LIN {X 0,Y 234.885,Z 274.225,A -85,B 0,C 180,E1 -19755.899,E2 -19755.899} C_VEL
LIN {X 0,Y 234.884,Z 274.226,A -85,B 0,C 180,E1 -19758.832,E2 -19758.832} C_VEL
LIN {X 0,Y 234.922,Z 274.22,A -85,B 0,C 180,E1 -19761.079,E2 -19761.079} C_VEL
LIN {X 0,Y 234.962,Z 274.217,A -85,B 0,C 180,E1 -19765.367,E2 -19765.367} C_VEL
LIN {X 0,Y 234.972,Z 274.217,A -85,B 0,C 180,E1 -19770.157,E2 -19770.157} C_VEL
LIN {X 0,Y 234.997,Z 274.213,A -85,B 0,C 180,E1 -19773.794,E2 -19773.794} C_VEL
LIN {X 0,Y 234.993,Z 274.213,A -85,B 0,C 180,E1 -19778.968,E2 -19778.968} C_VEL
LIN {X 0,Y 235.066,Z 274.203,A -85,B 0,C 180,E1 -19783.086,E2 -19783.086} C_VEL
LIN {X 0,Y 235.112,Z 274.196,A -85,B 0,C 180,E1 -19787.922,E2 -19787.922} C_VEL
LIN {X 0,Y 235.325,Z 274.173,A -85,B 0,C 180,E1 -19791.412,E2 -19791.412} C_VEL
LIN {X 0,Y 235.361,Z 274.167,A -85,B 0,C 180,E1 -19793.14,E2 -19793.14} C_VEL
LIN {X 0,Y 235.581,Z 274.14,A -85,B 0,C 180,E1 -19798.29,E2 -19798.29} C_VEL
LIN {X 0,Y 235.598,Z 274.136,A -85,B 0,C 180,E1 -19801.709,E2 -19801.709} C_VEL
LIN {X 0,Y 235.37,Z 274.166,A -85,B 0,C 180,E1 -19806.86,E2 -19806.86} C_VEL
LIN {X 0,Y 235.217,Z 274.185,A -85,B 0,C 180,E1 -19810.327,E2 -19810.327} C_VEL
LIN {X 0,Y 235.116,Z 274.196,A -85,B 0,C 180,E1 -19815.606,E2 -19815.606} C_VEL
LIN {X 0,Y 235.01,Z 274.209,A -85,B 0,C 180,E1 -19819.205,E2 -19819.205} C_VEL
LIN {X 0,Y 234.942,Z 274.219,A -85,B 0,C 180,E1 -19822.885,E2 -19822.885} C_VEL
LIN {X 0,Y 234.931,Z 274.22,A -85,B 0,C 180,E1 -19826.662,E2 -19826.662} C_VEL
LIN {X 0,Y 234.9,Z 274.225,A -85,B 0,C 180,E1 -19830.572,E2 -19830.572} C_VEL
LIN {X 0,Y 234.927,Z 274.224,A -85,B 0,C 180,E1 -19834.639,E2 -19834.639} C_VEL
LIN {X 0,Y 234.963,Z 274.311,A -85,B 0,C 180,E1 -19838.638,E2 -19838.638} C_VEL
LIN {X 0,Y 235.52,Z 277.972,A -85,B 0,C 180,E1 -19843.34,E2 -19843.34} C_VEL
LIN {X 0,Y 236.021,Z 280.862,A -85,B 0,C 180,E1 -19846.774,E2 -19846.774} C_VEL
LIN {X 0,Y 236.594,Z 284.553,A -85,B 0,C 180,E1 -19850.896,E2 -19850.896} C_VEL
LIN {X 0,Y 235.974,Z 285.513,A -85,B 0,C 180,E1 -19851.81,E2 -19851.81} C_VEL
LIN {X 0,Y 233.129,Z 287.277,A -85,B 0,C 180,E1 -19853.227,E2 -19853.227} C_VEL
LIN {X 0,Y 230.118,Z 289.077,A -85,B 0,C 180,E1 -19854.673,E2 -19854.673} C_VEL
LIN {X 0,Y 229.294,Z 290.098,A -85,B 0,C 180,E1 -19855.624,E2 -19855.624} C_VEL
LIN {X 0,Y 228.939,Z 291.784,A -85,B 0,C 180,E1 -19857.204,E2 -19857.204} C_VEL
LIN {X 0,Y 229.832,Z 294.982,A -85,B 0,C 180,E1 -19857.512,E2 -19857.512} C_VEL
LIN {X 0,Y 233.461,Z 307.701,A -85,B 0,C 180,E1 -19858.946,E2 -19858.946} C_VEL
LIN {X 0,Y 235.843,Z 319.474,A -85,B 0,C 180,E1 -19860.432,E2 -19860.432} C_VEL
LIN {X 0,Y 237.308,Z 330.805,A -85,B 0,C 180,E1 -19862.06,E2 -19862.06} C_VEL
LIN {X 0,Y 237.836,Z 342.077,A -85,B 0,C 180,E1 -19863.924,E2 -19863.924} C_VEL
LIN {X 0,Y 237.611,Z 348.307,A -85,B 0,C 180,E1 -19865.071,E2 -19865.071} C_VEL
LIN {X 0,Y 234.977,Z 358.761,A -85,B 0,C 180,E1 -19867.119,E2 -19867.119} C_VEL
LIN {X 0,Y 232.724,Z 367.292,A -85,B 0,C 180,E1 -19869.237,E2 -19869.237} C_VEL
LIN {X 0,Y 230.624,Z 375.499,A -85,B 0,C 180,E1 -19871.798,E2 -19871.798} C_VEL
LIN {X 0,Y 228.803,Z 382.165,A -85,B 0,C 180,E1 -19874.409,E2 -19874.409} C_VEL
LIN {X 0,Y 227.207,Z 388.266,A -85,B 0,C 180,E1 -19877.495,E2 -19877.495} C_VEL
LIN {X 0,Y 226.332,Z 392.236,A -85,B 0,C 180,E1 -19880.166,E2 -19880.166} C_VEL
LIN {X 0,Y 225.809,Z 395.171,A -85,B 0,C 180,E1 -19882.848,E2 -19882.848} C_VEL
LIN {X 0,Y 225.59,Z 397.12,A -85,B 0,C 180,E1 -19885.505,E2 -19885.505} C_VEL
LIN {X 0,Y 225.644,Z 398.178,A -85,B 0,C 180,E1 -19888.215,E2 -19888.215} C_VEL
LIN {X 0,Y 225.716,Z 398.393,A -85,B 0,C 180,E1 -19890,E2 -19890} C_VEL
LIN {X 0,Y 225.642,Z 398.168,A -85,B 0,C 180,E1 -19891.785,E2 -19891.785} C_VEL
LIN {X 0,Y 225.643,Z 396.545,A -85,B 0,C 180,E1 -19895.361,E2 -19895.361} C_VEL
LIN {X 0,Y 225.779,Z 395.136,A -85,B 0,C 180,E1 -19897.152,E2 -19897.152} C_VEL
LIN {X 0,Y 226.332,Z 392.186,A -85,B 0,C 180,E1 -19899.833,E2 -19899.833} C_VEL
LIN {X 0,Y 227.206,Z 388.196,A -85,B 0,C 180,E1 -19902.505,E2 -19902.505} C_VEL
LIN {X 0,Y 228.797,Z 382.068,A -85,B 0,C 180,E1 -19905.591,E2 -19905.591} C_VEL
LIN {X 0,Y 230.624,Z 375.38,A -85,B 0,C 180,E1 -19908.201,E2 -19908.201} C_VEL
LIN {X 0,Y 232.613,Z 368.002,A -85,B 0,C 180,E1 -19910.509,E2 -19910.509} C_VEL
LIN {X 0,Y 235.015,Z 358.578,A -85,B 0,C 180,E1 -19912.877,E2 -19912.877} C_VEL
LIN {X 0,Y 237.592,Z 348.074,A -85,B 0,C 180,E1 -19914.93,E2 -19914.93} C_VEL
LIN {X 0,Y 237.692,Z 338.928,A -85,B 0,C 180,E1 -19916.585,E2 -19916.585} C_VEL
LIN {X 0,Y 237.116,Z 329.199,A -85,B 0,C 180,E1 -19918.134,E2 -19918.134} C_VEL
LIN {X 0,Y 235.415,Z 317.231,A -85,B 0,C 180,E1 -19919.816,E2 -19919.816} C_VEL
LIN {X 0,Y 232.586,Z 304.36,A -85,B 0,C 180,E1 -19921.403,E2 -19921.403} C_VEL
LIN {X 0,Y 229.458,Z 294.179,A -85,B 0,C 180,E1 -19922.535,E2 -19922.535} C_VEL
LIN {X 0,Y 228.907,Z 291.66,A -85,B 0,C 180,E1 -19922.767,E2 -19922.767} C_VEL
LIN {X 0,Y 229.544,Z 288.869,A -85,B 0,C 180,E1 -19925.572,E2 -19925.572} C_VEL
LIN {X 0,Y 229.598,Z 285.783,A -85,B 0,C 180,E1 -19928.866,E2 -19928.866} C_VEL
LIN {X 0,Y 229.109,Z 282.514,A -85,B 0,C 180,E1 -19932.591,E2 -19932.591} C_VEL
LIN {X 0,Y 228.398,Z 278.449,A -85,B 0,C 180,E1 -19937.604,E2 -19937.604} C_VEL
LIN {X 0,Y 227.922,Z 275.092,A -85,B 0,C 180,E1 -19942.314,E2 -19942.314} C_VEL
LIN {X 0,Y 227.879,Z 275.104,A -85,B 0,C 180,E1 -19946.378,E2 -19946.378} C_VEL
LIN {X 0,Y 227.876,Z 275.105,A -85,B 0,C 180,E1 -19950.432,E2 -19950.432} C_VEL
LIN {X 0,Y 227.881,Z 275.103,A -85,B 0,C 180,E1 -19954.42,E2 -19954.42} C_VEL
LIN {X 0,Y 227.952,Z 275.092,A -85,B 0,C 180,E1 -19958.286,E2 -19958.286} C_VEL
LIN {X 0,Y 228.035,Z 275.079,A -85,B 0,C 180,E1 -19962.826,E2 -19962.826} C_VEL
LIN {X 0,Y 228.073,Z 275.075,A -85,B 0,C 180,E1 -19967.543,E2 -19967.543} C_VEL
LIN {X 0,Y 228.265,Z 275.052,A -85,B 0,C 180,E1 -19971.144,E2 -19971.144} C_VEL
LIN {X 0,Y 228.32,Z 275.043,A -85,B 0,C 180,E1 -19972.928,E2 -19972.928} C_VEL
LIN {X 0,Y 228.555,Z 275.011,A -85,B 0,C 180,E1 -19978.238,E2 -19978.238} C_VEL
LIN {X 0,Y 228.54,Z 275.015,A -85,B 0,C 180,E1 -19981.762,E2 -19981.762} C_VEL
LIN {X 0,Y 228.315,Z 275.046,A -85,B 0,C 180,E1 -19987.073,E2 -19987.073} C_VEL
LIN {X 0,Y 228.143,Z 275.068,A -85,B 0,C 180,E1 -19990.651,E2 -19990.651} C_VEL
LIN {X 0,Y 228.042,Z 275.079,A -85,B 0,C 180,E1 -19994.274,E2 -19994.274} C_VEL
LIN {X 0,Y 227.97,Z 275.087,A -85,B 0,C 180,E1 -19997.956,E2 -19997.956} C_VEL
LIN {X 0,Y 227.917,Z 275.095,A -85,B 0,C 180,E1 -20002.32,E2 -20002.32} C_VEL
LIN {X 0,Y 227.945,Z 275.091,A -85,B 0,C 180,E1 -20006.603,E2 -20006.603} C_VEL
LIN {X 0,Y 227.911,Z 275.097,A -85,B 0,C 180,E1 -20010.297,E2 -20010.297} C_VEL
LIN {X 0,Y 227.89,Z 275.098,A -85,B 0,C 180,E1 -20013.719,E2 -20013.719} C_VEL
LIN {X 0,Y 227.849,Z 275.105,A -85,B 0,C 180,E1 -20018.09,E2 -20018.09} C_VEL
LIN {X 0,Y 227.806,Z 275.106,A -85,B 0,C 180,E1 -20022.744,E2 -20022.744} C_VEL
LIN {X 0,Y 227.793,Z 275.112,A -85,B 0,C 180,E1 -20027.253,E2 -20027.253} C_VEL
LIN {X 0,Y 227.794,Z 275.111,A -85,B 0,C 180,E1 -20027.771,E2 -20027.771} C_VEL
LIN {X 0,Y 228.121,Z 277.722,A -85,B 0,C 180,E1 -20031.963,E2 -20031.963} C_VEL
LIN {X 0,Y 228.132,Z 279.267,A -85,B 0,C 180,E1 -20034.174,E2 -20034.174} C_VEL
LIN {X 0,Y 227.974,Z 281.488,A -85,B 0,C 180,E1 -20037.173,E2 -20037.173} C_VEL
LIN {X 0,Y 229.009,Z 284.65,A -85,B 0,C 180,E1 -20037.516,E2 -20037.516} C_VEL
LIN {X 0,Y 233.392,Z 296.608,A -85,B 0,C 180,E1 -20039.049,E2 -20039.049} C_VEL
LIN {X 0,Y 236.369,Z 307.22,A -85,B 0,C 180,E1 -20040.527,E2 -20040.527} C_VEL
LIN {X 0,Y 238.446,Z 317.934,A -85,B 0,C 180,E1 -20042.157,E2 -20042.157} C_VEL
LIN {X 0,Y 239.698,Z 328.159,A -85,B 0,C 180,E1 -20043.909,E2 -20043.909} C_VEL
LIN {X 0,Y 239.776,Z 330.767,A -85,B 0,C 180,E1 -20044.384,E2 -20044.384} C_VEL
LIN {X 0,Y 237.493,Z 341.214,A -85,B 0,C 180,E1 -20046.223,E2 -20046.223} C_VEL
LIN {X 0,Y 235.276,Z 350.46,A -85,B 0,C 180,E1 -20048.263,E2 -20048.263} C_VEL
LIN {X 0,Y 232.951,Z 358.989,A -85,B 0,C 180,E1 -20050.618,E2 -20050.618} C_VEL
LIN {X 0,Y 230.753,Z 366.396,A -85,B 0,C 180,E1 -20053.182,E2 -20053.182} C_VEL
LIN {X 0,Y 229.031,Z 372.336,A -85,B 0,C 180,E1 -20055.79,E2 -20055.79} C_VEL
LIN {X 0,Y 227.7,Z 377.028,A -85,B 0,C 180,E1 -20058.427,E2 -20058.427} C_VEL
LIN {X 0,Y 226.773,Z 380.616,A -85,B 0,C 180,E1 -20061.086,E2 -20061.086} C_VEL
LIN {X 0,Y 226.101,Z 383.466,A -85,B 0,C 180,E1 -20064.086,E2 -20064.086} C_VEL
LIN {X 0,Y 225.853,Z 384.85,A -85,B 0,C 180,E1 -20066.432,E2 -20066.432} C_VEL
LIN {X 0,Y 225.747,Z 385.686,A -85,B 0,C 180,E1 -20070,E2 -20070} C_VEL
LIN {X 0,Y 225.75,Z 385.493,A -85,B 0,C 180,E1 -20071.784,E2 -20071.784} C_VEL
LIN {X 0,Y 225.853,Z 384.907,A -85,B 0,C 180,E1 -20073.568,E2 -20073.568} C_VEL
LIN {X 0,Y 226.335,Z 382.583,A -85,B 0,C 180,E1 -20077.135,E2 -20077.135} C_VEL
LIN {X 0,Y 227.072,Z 379.715,A -85,B 0,C 180,E1 -20079.801,E2 -20079.801} C_VEL
LIN {X 0,Y 228.089,Z 375.825,A -85,B 0,C 180,E1 -20082.456,E2 -20082.456} C_VEL
LIN {X 0,Y 229.547,Z 370.804,A -85,B 0,C 180,E1 -20085.085,E2 -20085.085} C_VEL
LIN {X 0,Y 231.365,Z 364.48,A -85,B 0,C 180,E1 -20087.684,E2 -20087.684} C_VEL
LIN {X 0,Y 233.685,Z 356.561,A -85,B 0,C 180,E1 -20090.234,E2 -20090.234} C_VEL
LIN {X 0,Y 235.646,Z 349.088,A -85,B 0,C 180,E1 -20092.195,E2 -20092.195} C_VEL
LIN {X 0,Y 237.852,Z 339.709,A -85,B 0,C 180,E1 -20094.204,E2 -20094.204} C_VEL
LIN {X 0,Y 239.901,Z 330.235,A -85,B 0,C 180,E1 -20095.835,E2 -20095.835} C_VEL
LIN {X 0,Y 238.792,Z 319.781,A -85,B 0,C 180,E1 -20097.674,E2 -20097.674} C_VEL
LIN {X 0,Y 236.677,Z 308.483,A -85,B 0,C 180,E1 -20099.435,E2 -20099.435} C_VEL
LIN {X 0,Y 234.207,Z 299.118,A -85,B 0,C 180,E1 -20100.756,E2 -20100.756} C_VEL
LIN {X 0,Y 230.069,Z 287.427,A -85,B 0,C 180,E1 -20102.302,E2 -20102.302} C_VEL
LIN {X 0,Y 227.94,Z 281.449,A -85,B 0,C 180,E1 -20103.022,E2 -20103.022} C_VEL
LIN {X 0,Y 228.147,Z 278.702,A -85,B 0,C 180,E1 -20106.781,E2 -20106.781} C_VEL
LIN {X 0,Y 227.963,Z 276.309,A -85,B 0,C 180,E1 -20110.348,E2 -20110.348} C_VEL
LIN {X 0,Y 227.796,Z 275.113,A -85,B 0,C 180,E1 -20112.23,E2 -20112.23} C_VEL
LIN {X 0,Y 227.824,Z 275.102,A -85,B 0,C 180,E1 -20115.196,E2 -20115.196} C_VEL
LIN {X 0,Y 227.827,Z 275.105,A -85,B 0,C 180,E1 -20119.623,E2 -20119.623} C_VEL
LIN {X 0,Y 227.901,Z 275.098,A -85,B 0,C 180,E1 -20124.132,E2 -20124.132} C_VEL
LIN {X 0,Y 227.874,Z 275.097,A -85,B 0,C 180,E1 -20128.378,E2 -20128.378} C_VEL
LIN {X 0,Y 227.888,Z 275.094,A -85,B 0,C 180,E1 -20132.445,E2 -20132.445} C_VEL
LIN {X 0,Y 227.909,Z 275.09,A -85,B 0,C 180,E1 -20136.367,E2 -20136.367} C_VEL
LIN {X 0,Y 227.927,Z 275.092,A -85,B 0,C 180,E1 -20140.173,E2 -20140.173} C_VEL
LIN {X 0,Y 228.032,Z 275.08,A -85,B 0,C 180,E1 -20143.896,E2 -20143.896} C_VEL
LIN {X 0,Y 228.069,Z 275.075,A -85,B 0,C 180,E1 -20147.543,E2 -20147.543} C_VEL
LIN {X 0,Y 228.263,Z 275.052,A -85,B 0,C 180,E1 -20151.144,E2 -20151.144} C_VEL
LIN {X 0,Y 228.313,Z 275.046,A -85,B 0,C 180,E1 -20152.927,E2 -20152.927} C_VEL
LIN {X 0,Y 228.54,Z 275.017,A -85,B 0,C 180,E1 -20158.238,E2 -20158.238} C_VEL
LIN {X 0,Y 228.556,Z 275.013,A -85,B 0,C 180,E1 -20161.762,E2 -20161.762} C_VEL
LIN {X 0,Y 228.321,Z 275.043,A -85,B 0,C 180,E1 -20167.072,E2 -20167.072} C_VEL
LIN {X 0,Y 228.148,Z 275.067,A -85,B 0,C 180,E1 -20170.651,E2 -20170.651} C_VEL
LIN {X 0,Y 228.067,Z 275.077,A -85,B 0,C 180,E1 -20174.272,E2 -20174.272} C_VEL
LIN {X 0,Y 228.005,Z 275.083,A -85,B 0,C 180,E1 -20177.953,E2 -20177.953} C_VEL
LIN {X 0,Y 227.92,Z 275.095,A -85,B 0,C 180,E1 -20182.321,E2 -20182.321} C_VEL
LIN {X 0,Y 227.908,Z 275.094,A -85,B 0,C 180,E1 -20186.584,E2 -20186.584} C_VEL
LIN {X 0,Y 227.875,Z 275.101,A -85,B 0,C 180,E1 -20190.28,E2 -20190.28} C_VEL
LIN {X 0,Y 227.878,Z 275.102,A -85,B 0,C 180,E1 -20193.72,E2 -20193.72} C_VEL
LIN {X 0,Y 227.952,Z 275.294,A -85,B 0,C 180,E1 -20198.07,E2 -20198.07} C_VEL
LIN {X 0,Y 228.451,Z 278.676,A -85,B 0,C 180,E1 -20202.594,E2 -20202.594} C_VEL
LIN {X 0,Y 228.782,Z 280.62,A -85,B 0,C 180,E1 -20205.045,E2 -20205.045} C_VEL
LIN {X 0,Y 229.307,Z 283.762,A -85,B 0,C 180,E1 -20208.78,E2 -20208.78} C_VEL
LIN {X 0,Y 229.621,Z 286.876,A -85,B 0,C 180,E1 -20212.255,E2 -20212.255} C_VEL
LIN {X 0,Y 229.555,Z 288.921,A -85,B 0,C 180,E1 -20214.43,E2 -20214.43} C_VEL
LIN {X 0,Y 229.294,Z 290.098,A -85,B 0,C 180,E1 -20215.624,E2 -20215.624} C_VEL
LIN {X 0,Y 229.334,Z 291.506,A -85,B 0,C 180,E1 -20216.361,E2 -20216.361} C_VEL
LIN {X 0,Y 229.683,Z 294.528,A -85,B 0,C 180,E1 -20217.107,E2 -20217.107} C_VEL
LIN {X 0,Y 230.101,Z 299.741,A -85,B 0,C 180,E1 -20217.804,E2 -20217.804} C_VEL
LIN {X 0,Y 229.759,Z 306.045,A -85,B 0,C 180,E1 -20218.259,E2 -20218.259} C_VEL
LIN {X 0,Y 228.821,Z 314.395,A -85,B 0,C 180,E1 -20218.89,E2 -20218.89} C_VEL
LIN {X 0,Y 228.994,Z 318.121,A -85,B 0,C 180,E1 -20219.328,E2 -20219.328} C_VEL
LIN {X 0,Y 230.539,Z 329.644,A -85,B 0,C 180,E1 -20221.03,E2 -20221.03} C_VEL
LIN {X 0,Y 231.175,Z 340.556,A -85,B 0,C 180,E1 -20222.869,E2 -20222.869} C_VEL
LIN {X 0,Y 231.134,Z 348.109,A -85,B 0,C 180,E1 -20224.323,E2 -20224.323} C_VEL
LIN {X 0,Y 228.449,Z 358.564,A -85,B 0,C 180,E1 -20226.426,E2 -20226.426} C_VEL
LIN {X 0,Y 225.753,Z 368.275,A -85,B 0,C 180,E1 -20228.943,E2 -20228.943} C_VEL
LIN {X 0,Y 223.867,Z 375.3,A -85,B 0,C 180,E1 -20231.229,E2 -20231.229} C_VEL
LIN {X 0,Y 221.929,Z 381.966,A -85,B 0,C 180,E1 -20233.913,E2 -20233.913} C_VEL
LIN {X 0,Y 220.226,Z 388.066,A -85,B 0,C 180,E1 -20237.092,E2 -20237.092} C_VEL
LIN {X 0,Y 219.318,Z 392.036,A -85,B 0,C 180,E1 -20239.849,E2 -20239.849} C_VEL
LIN {X 0,Y 218.736,Z 394.971,A -85,B 0,C 180,E1 -20242.616,E2 -20242.616} C_VEL
LIN {X 0,Y 218.488,Z 397.091,A -85,B 0,C 180,E1 -20245.685,E2 -20245.685} C_VEL
LIN {X 0,Y 218.541,Z 397.979,A -85,B 0,C 180,E1 -20248.157,E2 -20248.157} C_VEL
LIN {X 0,Y 218.631,Z 398.194,A -85,B 0,C 180,E1 -20250,E2 -20250} C_VEL
LIN {X 0,Y 218.539,Z 397.968,A -85,B 0,C 180,E1 -20251.843,E2 -20251.843} C_VEL
LIN {X 0,Y 218.484,Z 397.08,A -85,B 0,C 180,E1 -20254.302,E2 -20254.302} C_VEL
LIN {X 0,Y 218.709,Z 394.935,A -85,B 0,C 180,E1 -20257.385,E2 -20257.385} C_VEL
LIN {X 0,Y 219.317,Z 391.984,A -85,B 0,C 180,E1 -20260.151,E2 -20260.151} C_VEL
LIN {X 0,Y 220.226,Z 387.994,A -85,B 0,C 180,E1 -20262.908,E2 -20262.908} C_VEL
LIN {X 0,Y 221.922,Z 381.865,A -85,B 0,C 180,E1 -20266.087,E2 -20266.087} C_VEL
LIN {X 0,Y 223.873,Z 375.177,A -85,B 0,C 180,E1 -20268.77,E2 -20268.77} C_VEL
LIN {X 0,Y 226.172,Z 366.906,A -85,B 0,C 180,E1 -20271.407,E2 -20271.407} C_VEL
LIN {X 0,Y 228.459,Z 358.375,A -85,B 0,C 180,E1 -20273.573,E2 -20273.573} C_VEL
LIN {X 0,Y 231.076,Z 347.868,A -85,B 0,C 180,E1 -20275.684,E2 -20275.684} C_VEL
LIN {X 0,Y 231.009,Z 337.161,A -85,B 0,C 180,E1 -20277.682,E2 -20277.682} C_VEL
LIN {X 0,Y 230.172,Z 326.464,A -85,B 0,C 180,E1 -20279.414,E2 -20279.414} C_VEL
LIN {X 0,Y 228.497,Z 315.557,A -85,B 0,C 180,E1 -20280.978,E2 -20280.978} C_VEL
LIN {X 0,Y 225.642,Z 303.453,A -85,B 0,C 180,E1 -20282.537,E2 -20282.537} C_VEL
LIN {X 0,Y 222.241,Z 292.284,A -85,B 0,C 180,E1 -20283.822,E2 -20283.822} C_VEL
LIN {X 0,Y 222.151,Z 291.412,A -85,B 0,C 180,E1 -20283.927,E2 -20283.927} C_VEL
LIN {X 0,Y 222.571,Z 288.652,A -85,B 0,C 180,E1 -20286.866,E2 -20286.866} C_VEL
LIN {X 0,Y 222.562,Z 286.597,A -85,B 0,C 180,E1 -20289.165,E2 -20289.165} C_VEL
LIN {X 0,Y 221.977,Z 283.153,A -85,B 0,C 180,E1 -20293.264,E2 -20293.264} C_VEL
LIN {X 0,Y 221.325,Z 279.326,A -85,B 0,C 180,E1 -20298.176,E2 -20298.176} C_VEL
LIN {X 0,Y 220.864,Z 275.998,A -85,B 0,C 180,E1 -20302.866,E2 -20302.866} C_VEL
LIN {X 0,Y 220.812,Z 275.984,A -85,B 0,C 180,E1 -20307.243,E2 -20307.243} C_VEL
LIN {X 0,Y 220.801,Z 275.985,A -85,B 0,C 180,E1 -20311.481,E2 -20311.481} C_VEL
LIN {X 0,Y 220.833,Z 275.98,A -85,B 0,C 180,E1 -20315.561,E2 -20315.561} C_VEL
LIN {X 0,Y 220.884,Z 275.972,A -85,B 0,C 180,E1 -20319.513,E2 -20319.513} C_VEL
LIN {X 0,Y 221.017,Z 275.955,A -85,B 0,C 180,E1 -20323.37,E2 -20323.37} C_VEL
LIN {X 0,Y 221.012,Z 275.953,A -85,B 0,C 180,E1 -20327.139,E2 -20327.139} C_VEL
LIN {X 0,Y 221.203,Z 275.93,A -85,B 0,C 180,E1 -20330.859,E2 -20330.859} C_VEL
LIN {X 0,Y 221.138,Z 275.937,A -85,B 0,C 180,E1 -20334.529,E2 -20334.529} C_VEL
LIN {X 0,Y 221.513,Z 275.889,A -85,B 0,C 180,E1 -20338.182,E2 -20338.182} C_VEL
LIN {X 0,Y 221.474,Z 275.895,A -85,B 0,C 180,E1 -20341.819,E2 -20341.819} C_VEL
LIN {X 0,Y 221.252,Z 275.924,A -85,B 0,C 180,E1 -20347.3,E2 -20347.3} C_VEL
LIN {X 0,Y 221.064,Z 275.948,A -85,B 0,C 180,E1 -20350.997,E2 -20350.997} C_VEL
LIN {X 0,Y 220.992,Z 275.958,A -85,B 0,C 180,E1 -20356.632,E2 -20356.632} C_VEL
LIN {X 0,Y 220.877,Z 275.972,A -85,B 0,C 180,E1 -20360.488,E2 -20360.488} C_VEL
LIN {X 0,Y 220.863,Z 275.973,A -85,B 0,C 180,E1 -20364.436,E2 -20364.436} C_VEL
LIN {X 0,Y 220.839,Z 275.976,A -85,B 0,C 180,E1 -20368.513,E2 -20368.513} C_VEL
LIN {X 0,Y 220.825,Z 275.978,A -85,B 0,C 180,E1 -20372.755,E2 -20372.755} C_VEL
LIN {X 0,Y 220.839,Z 275.976,A -85,B 0,C 180,E1 -20377.288,E2 -20377.288} C_VEL
LIN {X 0,Y 220.768,Z 275.984,A -85,B 0,C 180,E1 -20381.953,E2 -20381.953} C_VEL
LIN {X 0,Y 220.763,Z 275.987,A -85,B 0,C 180,E1 -20385.543,E2 -20385.543} C_VEL
LIN {X 0,Y 220.751,Z 275.989,A -85,B 0,C 180,E1 -20387.075,E2 -20387.075} C_VEL
LIN {X 0,Y 221.057,Z 277.949,A -85,B 0,C 180,E1 -20390.517,E2 -20390.517} C_VEL
LIN {X 0,Y 221.13,Z 279.485,A -85,B 0,C 180,E1 -20392.853,E2 -20392.853} C_VEL
LIN {X 0,Y 221.021,Z 281.838,A -85,B 0,C 180,E1 -20396.007,E2 -20396.007} C_VEL
LIN {X 0,Y 222.261,Z 285.131,A -85,B 0,C 180,E1 -20396.415,E2 -20396.415} C_VEL
LIN {X 0,Y 226.389,Z 296.266,A -85,B 0,C 180,E1 -20397.93,E2 -20397.93} C_VEL
LIN {X 0,Y 229.522,Z 306.734,A -85,B 0,C 180,E1 -20399.475,E2 -20399.475} C_VEL
LIN {X 0,Y 231.762,Z 318.117,A -85,B 0,C 180,E1 -20401.276,E2 -20401.276} C_VEL
LIN {X 0,Y 233.027,Z 328.374,A -85,B 0,C 180,E1 -20403.103,E2 -20403.103} C_VEL
LIN {X 0,Y 233.117,Z 332.258,A -85,B 0,C 180,E1 -20403.838,E2 -20403.838} C_VEL
LIN {X 0,Y 230.757,Z 342.47,A -85,B 0,C 180,E1 -20405.722,E2 -20405.722} C_VEL
LIN {X 0,Y 228.615,Z 350.944,A -85,B 0,C 180,E1 -20407.676,E2 -20407.676} C_VEL
LIN {X 0,Y 226.266,Z 359.191,A -85,B 0,C 180,E1 -20410.022,E2 -20410.022} C_VEL
LIN {X 0,Y 223.971,Z 366.597,A -85,B 0,C 180,E1 -20412.657,E2 -20412.657} C_VEL
LIN {X 0,Y 222.157,Z 372.537,A -85,B 0,C 180,E1 -20415.34,E2 -20415.34} C_VEL
LIN {X 0,Y 220.745,Z 377.229,A -85,B 0,C 180,E1 -20418.057,E2 -20418.057} C_VEL
LIN {X 0,Y 219.773,Z 380.817,A -85,B 0,C 180,E1 -20420.8,E2 -20420.8} C_VEL
LIN {X 0,Y 219,Z 383.876,A -85,B 0,C 180,E1 -20424.174,E2 -20424.174} C_VEL
LIN {X 0,Y 218.765,Z 385.05,A -85,B 0,C 180,E1 -20426.316,E2 -20426.316} C_VEL
LIN {X 0,Y 218.67,Z 385.657,A -85,B 0,C 180,E1 -20428.158,E2 -20428.158} C_VEL
LIN {X 0,Y 218.662,Z 385.885,A -85,B 0,C 180,E1 -20430,E2 -20430} C_VEL
LIN {X 0,Y 218.67,Z 385.692,A -85,B 0,C 180,E1 -20431.842,E2 -20431.842} C_VEL
LIN {X 0,Y 218.765,Z 385.106,A -85,B 0,C 180,E1 -20433.684,E2 -20433.684} C_VEL
LIN {X 0,Y 219.045,Z 383.886,A -85,B 0,C 180,E1 -20435.939,E2 -20435.939} C_VEL
LIN {X 0,Y 219.783,Z 380.969,A -85,B 0,C 180,E1 -20439.2,E2 -20439.2} C_VEL
LIN {X 0,Y 220.718,Z 377.438,A -85,B 0,C 180,E1 -20441.945,E2 -20441.945} C_VEL
LIN {X 0,Y 222.13,Z 372.802,A -85,B 0,C 180,E1 -20444.662,E2 -20444.662} C_VEL
LIN {X 0,Y 224.248,Z 365.812,A -85,B 0,C 180,E1 -20447.793,E2 -20447.793} C_VEL
LIN {X 0,Y 226.609,Z 358.229,A -85,B 0,C 180,E1 -20450.421,E2 -20450.421} C_VEL
LIN {X 0,Y 228.953,Z 349.809,A -85,B 0,C 180,E1 -20452.739,E2 -20452.739} C_VEL
LIN {X 0,Y 231.384,Z 339.905,A -85,B 0,C 180,E1 -20454.926,E2 -20454.926} C_VEL
LIN {X 0,Y 233.29,Z 331.717,A -85,B 0,C 180,E1 -20456.382,E2 -20456.382} C_VEL
LIN {X 0,Y 232.431,Z 322.328,A -85,B 0,C 180,E1 -20458.131,E2 -20458.131} C_VEL
LIN {X 0,Y 230.553,Z 311.378,A -85,B 0,C 180,E1 -20459.958,E2 -20459.958} C_VEL
LIN {X 0,Y 228.018,Z 301.264,A -85,B 0,C 180,E1 -20461.49,E2 -20461.49} C_VEL
LIN {X 0,Y 223.748,Z 288.775,A -85,B 0,C 180,E1 -20463.25,E2 -20463.25} C_VEL
LIN {X 0,Y 221.095,Z 282.49,A -85,B 0,C 180,E1 -20464.1,E2 -20464.1} C_VEL
LIN {X 0,Y 220.947,Z 281.662,A -85,B 0,C 180,E1 -20464.206,E2 -20464.206} C_VEL
LIN {X 0,Y 221.134,Z 279.434,A -85,B 0,C 180,E1 -20467.388,E2 -20467.388} C_VEL
LIN {X 0,Y 220.985,Z 277.582,A -85,B 0,C 180,E1 -20470.246,E2 -20470.246} C_VEL
LIN {X 0,Y 220.752,Z 275.981,A -85,B 0,C 180,E1 -20472.925,E2 -20472.925} C_VEL
LIN {X 0,Y 220.763,Z 275.985,A -85,B 0,C 180,E1 -20477.072,E2 -20477.072} C_VEL
LIN {X 0,Y 220.808,Z 275.98,A -85,B 0,C 180,E1 -20480.463,E2 -20480.463} C_VEL
LIN {X 0,Y 220.826,Z 275.976,A -85,B 0,C 180,E1 -20482.793,E2 -20482.793} C_VEL
LIN {X 0,Y 220.826,Z 275.978,A -85,B 0,C 180,E1 -20487.245,E2 -20487.245} C_VEL
LIN {X 0,Y 220.839,Z 275.976,A -85,B 0,C 180,E1 -20491.487,E2 -20491.487} C_VEL
LIN {X 0,Y 220.865,Z 275.971,A -85,B 0,C 180,E1 -20495.565,E2 -20495.565} C_VEL
LIN {X 0,Y 220.879,Z 275.972,A -85,B 0,C 180,E1 -20499.512,E2 -20499.512} C_VEL
LIN {X 0,Y 220.993,Z 275.958,A -85,B 0,C 180,E1 -20503.368,E2 -20503.368} C_VEL
LIN {X 0,Y 221.068,Z 275.948,A -85,B 0,C 180,E1 -20509.004,E2 -20509.004} C_VEL
LIN {X 0,Y 221.25,Z 275.926,A -85,B 0,C 180,E1 -20512.7,E2 -20512.7} C_VEL
LIN {X 0,Y 221.473,Z 275.897,A -85,B 0,C 180,E1 -20518.181,E2 -20518.181} C_VEL
LIN {X 0,Y 221.514,Z 275.89,A -85,B 0,C 180,E1 -20521.818,E2 -20521.818} C_VEL
LIN {X 0,Y 221.257,Z 275.922,A -85,B 0,C 180,E1 -20527.299,E2 -20527.299} C_VEL
LIN {X 0,Y 221.07,Z 275.948,A -85,B 0,C 180,E1 -20530.996,E2 -20530.996} C_VEL
LIN {X 0,Y 220.998,Z 275.955,A -85,B 0,C 180,E1 -20534.739,E2 -20534.739} C_VEL
LIN {X 0,Y 220.923,Z 275.966,A -85,B 0,C 180,E1 -20538.549,E2 -20538.549} C_VEL
LIN {X 0,Y 220.866,Z 275.972,A -85,B 0,C 180,E1 -20542.662,E2 -20542.662} C_VEL
LIN {X 0,Y 220.854,Z 275.973,A -85,B 0,C 180,E1 -20546.999,E2 -20546.999} C_VEL
LIN {X 0,Y 220.82,Z 275.979,A -85,B 0,C 180,E1 -20550.758,E2 -20550.758} C_VEL
LIN {X 0,Y 220.795,Z 275.984,A -85,B 0,C 180,E1 -20554.956,E2 -20554.956} C_VEL
LIN {X 0,Y 220.894,Z 276.177,A -85,B 0,C 180,E1 -20557.306,E2 -20557.306} C_VEL
LIN {X 0,Y 221.348,Z 279.408,A -85,B 0,C 180,E1 -20561.818,E2 -20561.818} C_VEL
LIN {X 0,Y 221.988,Z 283.216,A -85,B 0,C 180,E1 -20566.733,E2 -20566.733} C_VEL
LIN {X 0,Y 222.562,Z 286.651,A -85,B 0,C 180,E1 -20570.835,E2 -20570.835} C_VEL
LIN {X 0,Y 222.54,Z 289.729,A -85,B 0,C 180,E1 -20574.251,E2 -20574.251} C_VEL
LIN {X 0,Y 222.147,Z 291.448,A -85,B 0,C 180,E1 -20576.055,E2 -20576.055} C_VEL
LIN {X 0,Y 223.067,Z 294.804,A -85,B 0,C 180,E1 -20576.401,E2 -20576.401} C_VEL
LIN {X 0,Y 226.676,Z 307.124,A -85,B 0,C 180,E1 -20577.876,E2 -20577.876} C_VEL
LIN {X 0,Y 228.994,Z 318.121,A -85,B 0,C 180,E1 -20579.328,E2 -20579.328} C_VEL
LIN {X 0,Y 229.149,Z 323.436,A -85,B 0,C 180,E1 -20579.988,E2 -20579.988} C_VEL
LIN {X 0,Y 227.421,Z 332.31,A -85,B 0,C 180,E1 -20581.007,E2 -20581.007} C_VEL
LIN {X 0,Y 225.179,Z 340.906,A -85,B 0,C 180,E1 -20582.173,E2 -20582.173} C_VEL
LIN {X 0,Y 224.568,Z 345.73,A -85,B 0,C 180,E1 -20583.054,E2 -20583.054} C_VEL
LIN {X 0,Y 224.196,Z 350.215,A -85,B 0,C 180,E1 -20583.968,E2 -20583.968} C_VEL
LIN {X 0,Y 221.402,Z 360.16,A -85,B 0,C 180,E1 -20586.126,E2 -20586.126} C_VEL
LIN {X 0,Y 218.657,Z 369.706,A -85,B 0,C 180,E1 -20588.766,E2 -20588.766} C_VEL
LIN {X 0,Y 216.748,Z 376.338,A -85,B 0,C 180,E1 -20591.08,E2 -20591.08} C_VEL
LIN {X 0,Y 214.811,Z 382.762,A -85,B 0,C 180,E1 -20593.853,E2 -20593.853} C_VEL
LIN {X 0,Y 213.261,Z 387.866,A -85,B 0,C 180,E1 -20596.662,E2 -20596.662} C_VEL
LIN {X 0,Y 212.304,Z 391.836,A -85,B 0,C 180,E1 -20599.509,E2 -20599.509} C_VEL
LIN {X 0,Y 211.67,Z 394.771,A -85,B 0,C 180,E1 -20602.368,E2 -20602.368} C_VEL
LIN {X 0,Y 211.393,Z 397.026,A -85,B 0,C 180,E1 -20605.855,E2 -20605.855} C_VEL
LIN {X 0,Y 211.442,Z 397.779,A -85,B 0,C 180,E1 -20608.095,E2 -20608.095} C_VEL
LIN {X 0,Y 211.547,Z 397.994,A -85,B 0,C 180,E1 -20610,E2 -20610} C_VEL
LIN {X 0,Y 211.44,Z 397.767,A -85,B 0,C 180,E1 -20611.905,E2 -20611.905} C_VEL
LIN {X 0,Y 211.487,Z 396.144,A -85,B 0,C 180,E1 -20615.721,E2 -20615.721} C_VEL
LIN {X 0,Y 211.65,Z 394.734,A -85,B 0,C 180,E1 -20617.633,E2 -20617.633} C_VEL
LIN {X 0,Y 212.304,Z 391.783,A -85,B 0,C 180,E1 -20620.49,E2 -20620.49} C_VEL
LIN {X 0,Y 213.26,Z 387.791,A -85,B 0,C 180,E1 -20623.337,E2 -20623.337} C_VEL
LIN {X 0,Y 215.085,Z 381.663,A -85,B 0,C 180,E1 -20626.613,E2 -20626.613} C_VEL
LIN {X 0,Y 217.151,Z 374.975,A -85,B 0,C 180,E1 -20629.374,E2 -20629.374} C_VEL
LIN {X 0,Y 219.43,Z 367.056,A -85,B 0,C 180,E1 -20631.981,E2 -20631.981} C_VEL
LIN {X 0,Y 221.962,Z 358.172,A -85,B 0,C 180,E1 -20634.307,E2 -20634.307} C_VEL
LIN {X 0,Y 224.422,Z 348.841,A -85,B 0,C 180,E1 -20636.253,E2 -20636.253} C_VEL
LIN {X 0,Y 224.461,Z 338.049,A -85,B 0,C 180,E1 -20638.367,E2 -20638.367} C_VEL
LIN {X 0,Y 223.681,Z 327.455,A -85,B 0,C 180,E1 -20640.18,E2 -20640.18} C_VEL
LIN {X 0,Y 221.863,Z 315.531,A -85,B 0,C 180,E1 -20641.988,E2 -20641.988} C_VEL
LIN {X 0,Y 218.944,Z 303.041,A -85,B 0,C 180,E1 -20643.676,E2 -20643.676} C_VEL
LIN {X 0,Y 215.359,Z 291.471,A -85,B 0,C 180,E1 -20645.084,E2 -20645.084} C_VEL
LIN {X 0,Y 215.543,Z 289.456,A -85,B 0,C 180,E1 -20647.1,E2 -20647.1} C_VEL
LIN {X 0,Y 215.335,Z 286.357,A -85,B 0,C 180,E1 -20650.749,E2 -20650.749} C_VEL
LIN {X 0,Y 214.875,Z 283.776,A -85,B 0,C 180,E1 -20653.982,E2 -20653.982} C_VEL
LIN {X 0,Y 214.277,Z 280.043,A -85,B 0,C 180,E1 -20659.006,E2 -20659.006} C_VEL
LIN {X 0,Y 213.79,Z 276.856,A -85,B 0,C 180,E1 -20663.83,E2 -20663.83} C_VEL
LIN {X 0,Y 213.768,Z 276.863,A -85,B 0,C 180,E1 -20668.737,E2 -20668.737} C_VEL
LIN {X 0,Y 213.784,Z 276.859,A -85,B 0,C 180,E1 -20672.597,E2 -20672.597} C_VEL
LIN {X 0,Y 213.808,Z 276.854,A -85,B 0,C 180,E1 -20676.981,E2 -20676.981} C_VEL
LIN {X 0,Y 213.944,Z 276.835,A -85,B 0,C 180,E1 -20682.804,E2 -20682.804} C_VEL
LIN {X 0,Y 213.954,Z 276.831,A -85,B 0,C 180,E1 -20686.707,E2 -20686.707} C_VEL
LIN {X 0,Y 214.141,Z 276.81,A -85,B 0,C 180,E1 -20690.555,E2 -20690.555} C_VEL
LIN {X 0,Y 214.099,Z 276.814,A -85,B 0,C 180,E1 -20694.349,E2 -20694.349} C_VEL
LIN {X 0,Y 214.446,Z 276.769,A -85,B 0,C 180,E1 -20698.122,E2 -20698.122} C_VEL
LIN {X 0,Y 214.541,Z 276.76,A -85,B 0,C 180,E1 -20700,E2 -20700} C_VEL
LIN {X 0,Y 214.411,Z 276.775,A -85,B 0,C 180,E1 -20701.878,E2 -20701.878} C_VEL
LIN {X 0,Y 214.192,Z 276.803,A -85,B 0,C 180,E1 -20707.542,E2 -20707.542} C_VEL
LIN {X 0,Y 213.995,Z 276.826,A -85,B 0,C 180,E1 -20711.365,E2 -20711.365} C_VEL
LIN {X 0,Y 213.91,Z 276.837,A -85,B 0,C 180,E1 -20715.239,E2 -20715.239} C_VEL
LIN {X 0,Y 213.82,Z 276.85,A -85,B 0,C 180,E1 -20719.189,E2 -20719.189} C_VEL
LIN {X 0,Y 213.812,Z 276.851,A -85,B 0,C 180,E1 -20723.231,E2 -20723.231} C_VEL
LIN {X 0,Y 213.83,Z 276.848,A -85,B 0,C 180,E1 -20727.45,E2 -20727.45} C_VEL
LIN {X 0,Y 213.78,Z 276.855,A -85,B 0,C 180,E1 -20731.736,E2 -20731.736} C_VEL
LIN {X 0,Y 213.749,Z 276.861,A -85,B 0,C 180,E1 -20736.288,E2 -20736.288} C_VEL
LIN {X 0,Y 213.712,Z 276.865,A -85,B 0,C 180,E1 -20741.126,E2 -20741.126} C_VEL
LIN {X 0,Y 213.704,Z 276.867,A -85,B 0,C 180,E1 -20743.68,E2 -20743.68} C_VEL
LIN {X 0,Y 213.702,Z 276.865,A -85,B 0,C 180,E1 -20746.345,E2 -20746.345} C_VEL
LIN {X 0,Y 213.93,Z 278.279,A -85,B 0,C 180,E1 -20749.077,E2 -20749.077} C_VEL
LIN {X 0,Y 214.106,Z 280.085,A -85,B 0,C 180,E1 -20751.981,E2 -20751.981} C_VEL
LIN {X 0,Y 214.038,Z 281.886,A -85,B 0,C 180,E1 -20754.701,E2 -20754.701} C_VEL
LIN {X 0,Y 215.214,Z 285.229,A -85,B 0,C 180,E1 -20755.15,E2 -20755.15} C_VEL
LIN {X 0,Y 218.702,Z 293.765,A -85,B 0,C 180,E1 -20756.407,E2 -20756.407} C_VEL
LIN {X 0,Y 222.22,Z 304.734,A -85,B 0,C 180,E1 -20758.091,E2 -20758.091} C_VEL
LIN {X 0,Y 224.483,Z 314.476,A -85,B 0,C 180,E1 -20759.68,E2 -20759.68} C_VEL
LIN {X 0,Y 226.04,Z 325.148,A -85,B 0,C 180,E1 -20761.583,E2 -20761.583} C_VEL
LIN {X 0,Y 226.625,Z 332.467,A -85,B 0,C 180,E1 -20763.029,E2 -20763.029} C_VEL
LIN {X 0,Y 224.298,Z 342.674,A -85,B 0,C 180,E1 -20764.976,E2 -20764.976} C_VEL
LIN {X 0,Y 221.912,Z 351.68,A -85,B 0,C 180,E1 -20767.125,E2 -20767.125} C_VEL
LIN {X 0,Y 219.195,Z 360.74,A -85,B 0,C 180,E1 -20769.838,E2 -20769.838} C_VEL
LIN {X 0,Y 216.85,Z 367.909,A -85,B 0,C 180,E1 -20772.555,E2 -20772.555} C_VEL
LIN {X 0,Y 215.302,Z 372.738,A -85,B 0,C 180,E1 -20774.862,E2 -20774.862} C_VEL
LIN {X 0,Y 213.797,Z 377.431,A -85,B 0,C 180,E1 -20777.663,E2 -20777.663} C_VEL
LIN {X 0,Y 212.752,Z 381.018,A -85,B 0,C 180,E1 -20780.493,E2 -20780.493} C_VEL
LIN {X 0,Y 212.244,Z 382.87,A -85,B 0,C 180,E1 -20782.389,E2 -20782.389} C_VEL
LIN {X 0,Y 211.893,Z 384.261,A -85,B 0,C 180,E1 -20784.29,E2 -20784.29} C_VEL
LIN {X 0,Y 211.592,Z 385.857,A -85,B 0,C 180,E1 -20788.097,E2 -20788.097} C_VEL
LIN {X 0,Y 211.579,Z 386.084,A -85,B 0,C 180,E1 -20790,E2 -20790} C_VEL
LIN {X 0,Y 211.592,Z 385.891,A -85,B 0,C 180,E1 -20791.904,E2 -20791.904} C_VEL
LIN {X 0,Y 211.893,Z 384.339,A -85,B 0,C 180,E1 -20795.711,E2 -20795.711} C_VEL
LIN {X 0,Y 212.245,Z 382.982,A -85,B 0,C 180,E1 -20797.611,E2 -20797.611} C_VEL
LIN {X 0,Y 213.058,Z 380.114,A -85,B 0,C 180,E1 -20800.453,E2 -20800.453} C_VEL
LIN {X 0,Y 214.223,Z 376.223,A -85,B 0,C 180,E1 -20803.277,E2 -20803.277} C_VEL
LIN {X 0,Y 215.844,Z 371.202,A -85,B 0,C 180,E1 -20806.067,E2 -20806.067} C_VEL
LIN {X 0,Y 217.894,Z 364.875,A -85,B 0,C 180,E1 -20808.817,E2 -20808.817} C_VEL
LIN {X 0,Y 220.431,Z 356.955,A -85,B 0,C 180,E1 -20811.51,E2 -20811.51} C_VEL
LIN {X 0,Y 222.701,Z 348.739,A -85,B 0,C 180,E1 -20813.768,E2 -20813.768} C_VEL
LIN {X 0,Y 225.227,Z 339.036,A -85,B 0,C 180,E1 -20815.904,E2 -20815.904} C_VEL
LIN {X 0,Y 226.7,Z 333.2,A -85,B 0,C 180,E1 -20816.962,E2 -20816.962} C_VEL
LIN {X 0,Y 225.904,Z 323.555,A -85,B 0,C 180,E1 -20818.853,E2 -20818.853} C_VEL
LIN {X 0,Y 224.108,Z 312.646,A -85,B 0,C 180,E1 -20820.771,E2 -20820.771} C_VEL
LIN {X 0,Y 221.973,Z 303.727,A -85,B 0,C 180,E1 -20822.215,E2 -20822.215} C_VEL
LIN {X 0,Y 217.702,Z 291.17,A -85,B 0,C 180,E1 -20824.13,E2 -20824.13} C_VEL
LIN {X 0,Y 214.939,Z 284.788,A -85,B 0,C 180,E1 -20825.087,E2 -20825.087} C_VEL
LIN {X 0,Y 213.996,Z 281.885,A -85,B 0,C 180,E1 -20825.478,E2 -20825.478} C_VEL
LIN {X 0,Y 214.077,Z 279.834,A -85,B 0,C 180,E1 -20828.591,E2 -20828.591} C_VEL
LIN {X 0,Y 213.917,Z 278.295,A -85,B 0,C 180,E1 -20831.078,E2 -20831.078} C_VEL
LIN {X 0,Y 213.704,Z 276.86,A -85,B 0,C 180,E1 -20833.68,E2 -20833.68} C_VEL
LIN {X 0,Y 213.705,Z 276.864,A -85,B 0,C 180,E1 -20836.345,E2 -20836.345} C_VEL
LIN {X 0,Y 213.736,Z 276.86,A -85,B 0,C 180,E1 -20841.336,E2 -20841.336} C_VEL
LIN {X 0,Y 213.77,Z 276.855,A -85,B 0,C 180,E1 -20846.02,E2 -20846.02} C_VEL
LIN {X 0,Y 213.783,Z 276.855,A -85,B 0,C 180,E1 -20850.454,E2 -20850.454} C_VEL
LIN {X 0,Y 213.801,Z 276.852,A -85,B 0,C 180,E1 -20854.701,E2 -20854.701} C_VEL
LIN {X 0,Y 213.8,Z 276.853,A -85,B 0,C 180,E1 -20858.802,E2 -20858.802} C_VEL
LIN {X 0,Y 213.924,Z 276.836,A -85,B 0,C 180,E1 -20862.802,E2 -20862.802} C_VEL
LIN {X 0,Y 213.946,Z 276.835,A -85,B 0,C 180,E1 -20866.706,E2 -20866.706} C_VEL
LIN {X 0,Y 214.14,Z 276.81,A -85,B 0,C 180,E1 -20870.555,E2 -20870.555} C_VEL
LIN {X 0,Y 214.086,Z 276.816,A -85,B 0,C 180,E1 -20874.348,E2 -20874.348} C_VEL
LIN {X 0,Y 214.41,Z 276.777,A -85,B 0,C 180,E1 -20878.122,E2 -20878.122} C_VEL
LIN {X 0,Y 214.517,Z 276.763,A -85,B 0,C 180,E1 -20880,E2 -20880} C_VEL
LIN {X 0,Y 214.447,Z 276.77,A -85,B 0,C 180,E1 -20881.878,E2 -20881.878} C_VEL
LIN {X 0,Y 214.197,Z 276.801,A -85,B 0,C 180,E1 -20887.541,E2 -20887.541} C_VEL
LIN {X 0,Y 214.001,Z 276.827,A -85,B 0,C 180,E1 -20891.364,E2 -20891.364} C_VEL
LIN {X 0,Y 213.936,Z 276.834,A -85,B 0,C 180,E1 -20895.237,E2 -20895.237} C_VEL
LIN {X 0,Y 213.839,Z 276.847,A -85,B 0,C 180,E1 -20899.187,E2 -20899.187} C_VEL
LIN {X 0,Y 213.801,Z 276.852,A -85,B 0,C 180,E1 -20903.232,E2 -20903.232} C_VEL
LIN {X 0,Y 213.786,Z 276.855,A -85,B 0,C 180,E1 -20907.426,E2 -20907.426} C_VEL
LIN {X 0,Y 213.76,Z 276.861,A -85,B 0,C 180,E1 -20911.739,E2 -20911.739} C_VEL
LIN {X 0,Y 213.795,Z 276.929,A -85,B 0,C 180,E1 -20916.278,E2 -20916.278} C_VEL
LIN {X 0,Y 214.295,Z 280.142,A -85,B 0,C 180,E1 -20921.035,E2 -20921.035} C_VEL
LIN {X 0,Y 214.895,Z 283.85,A -85,B 0,C 180,E1 -20926.013,E2 -20926.013} C_VEL
LIN {X 0,Y 215.343,Z 286.415,A -85,B 0,C 180,E1 -20929.252,E2 -20929.252} C_VEL
LIN {X 0,Y 215.549,Z 289.511,A -85,B 0,C 180,E1 -20932.901,E2 -20932.901} C_VEL
LIN {X 0,Y 215.353,Z 291.268,A -85,B 0,C 180,E1 -20934.838,E2 -20934.838} C_VEL
LIN {X 0,Y 216.336,Z 294.63,A -85,B 0,C 180,E1 -20935.211,E2 -20935.211} C_VEL
LIN {X 0,Y 219.824,Z 306.297,A -85,B 0,C 180,E1 -20936.693,E2 -20936.693} C_VEL
LIN {X 0,Y 222.377,Z 318.047,A -85,B 0,C 180,E1 -20938.327,E2 -20938.327} C_VEL
LIN {X 0,Y 223.936,Z 329.473,A -85,B 0,C 180,E1 -20940.095,E2 -20940.095} C_VEL
LIN {X 0,Y 224.575,Z 340.351,A -85,B 0,C 180,E1 -20942.003,E2 -20942.003} C_VEL
LIN {X 0,Y 224.568,Z 345.73,A -85,B 0,C 180,E1 -20943.054,E2 -20943.054} C_VEL
LIN {X 0,Y 224.06,Z 348.886,A -85,B 0,C 180,E1 -20943.661,E2 -20943.661} C_VEL
LIN {X 0,Y 222.041,Z 353.464,A -85,B 0,C 180,E1 -20944.469,E2 -20944.469} C_VEL
LIN {X 0,Y 215.086,Z 363.326,A -85,B 0,C 180,E1 -20946.356,E2 -20946.356} C_VEL
LIN {X 0,Y 212.764,Z 367.286,A -85,B 0,C 180,E1 -20947.382,E2 -20947.382} C_VEL
LIN {X 0,Y 212.286,Z 368.558,A -85,B 0,C 180,E1 -20947.772,E2 -20947.772} C_VEL
LIN {X 0,Y 210.027,Z 376.139,A -85,B 0,C 180,E1 -20950.45,E2 -20950.45} C_VEL
LIN {X 0,Y 207.953,Z 382.562,A -85,B 0,C 180,E1 -20953.305,E2 -20953.305} C_VEL
LIN {X 0,Y 206.314,Z 387.665,A -85,B 0,C 180,E1 -20956.205,E2 -20956.205} C_VEL
LIN {X 0,Y 205.283,Z 391.636,A -85,B 0,C 180,E1 -20959.146,E2 -20959.146} C_VEL
LIN {X 0,Y 204.626,Z 394.572,A -85,B 0,C 180,E1 -20962.103,E2 -20962.103} C_VEL
LIN {X 0,Y 204.398,Z 395.969,A -85,B 0,C 180,E1 -20964.079,E2 -20964.079} C_VEL
LIN {X 0,Y 204.345,Z 397.579,A -85,B 0,C 180,E1 -20968.029,E2 -20968.029} C_VEL
LIN {X 0,Y 204.465,Z 397.795,A -85,B 0,C 180,E1 -20970,E2 -20970} C_VEL
LIN {X 0,Y 204.343,Z 397.567,A -85,B 0,C 180,E1 -20971.971,E2 -20971.971} C_VEL
LIN {X 0,Y 204.394,Z 395.943,A -85,B 0,C 180,E1 -20975.921,E2 -20975.921} C_VEL
LIN {X 0,Y 204.611,Z 394.533,A -85,B 0,C 180,E1 -20977.897,E2 -20977.897} C_VEL
LIN {X 0,Y 205.282,Z 391.581,A -85,B 0,C 180,E1 -20980.853,E2 -20980.853} C_VEL
LIN {X 0,Y 206.313,Z 387.589,A -85,B 0,C 180,E1 -20983.795,E2 -20983.795} C_VEL
LIN {X 0,Y 208.279,Z 381.462,A -85,B 0,C 180,E1 -20987.173,E2 -20987.173} C_VEL
LIN {X 0,Y 210.46,Z 374.774,A -85,B 0,C 180,E1 -20990.016,E2 -20990.016} C_VEL
LIN {X 0,Y 212.897,Z 366.587,A -85,B 0,C 180,E1 -20992.784,E2 -20992.784} C_VEL
LIN {X 0,Y 215.48,Z 357.968,A -85,B 0,C 180,E1 -20995.087,E2 -20995.087} C_VEL
LIN {X 0,Y 217.776,Z 349.784,A -85,B 0,C 180,E1 -20996.859,E2 -20996.859} C_VEL
LIN {X 0,Y 217.952,Z 339.844,A -85,B 0,C 180,E1 -20998.926,E2 -20998.926} C_VEL
LIN {X 0,Y 217.288,Z 329.024,A -85,B 0,C 180,E1 -21000.894,E2 -21000.894} C_VEL
LIN {X 0,Y 215.86,Z 318.507,A -85,B 0,C 180,E1 -21002.601,E2 -21002.601} C_VEL
LIN {X 0,Y 213.167,Z 305.978,A -85,B 0,C 180,E1 -21004.433,E2 -21004.433} C_VEL
LIN {X 0,Y 209.678,Z 294.671,A -85,B 0,C 180,E1 -21005.976,E2 -21005.976} C_VEL
LIN {X 0,Y 208.547,Z 291.464,A -85,B 0,C 180,E1 -21006.397,E2 -21006.397} C_VEL
LIN {X 0,Y 208.488,Z 290.981,A -85,B 0,C 180,E1 -21006.481,E2 -21006.481} C_VEL
LIN {X 0,Y 208.383,Z 288.17,A -85,B 0,C 180,E1 -21009.852,E2 -21009.852} C_VEL
LIN {X 0,Y 208.054,Z 286.112,A -85,B 0,C 180,E1 -21012.5,E2 -21012.5} C_VEL
LIN {X 0,Y 207.444,Z 282.527,A -85,B 0,C 180,E1 -21017.345,E2 -21017.345} C_VEL
LIN {X 0,Y 206.977,Z 279.176,A -85,B 0,C 180,E1 -21022.324,E2 -21022.324} C_VEL
LIN {X 0,Y 206.729,Z 277.737,A -85,B 0,C 180,E1 -21024.694,E2 -21024.694} C_VEL
LIN {X 0,Y 206.695,Z 277.743,A -85,B 0,C 180,E1 -21029.334,E2 -21029.334} C_VEL
LIN {X 0,Y 206.696,Z 277.744,A -85,B 0,C 180,E1 -21033.767,E2 -21033.767} C_VEL
LIN {X 0,Y 206.734,Z 277.735,A -85,B 0,C 180,E1 -21038.041,E2 -21038.041} C_VEL
LIN {X 0,Y 206.873,Z 277.716,A -85,B 0,C 180,E1 -21042.197,E2 -21042.197} C_VEL
LIN {X 0,Y 206.896,Z 277.711,A -85,B 0,C 180,E1 -21046.244,E2 -21046.244} C_VEL
LIN {X 0,Y 207.1,Z 277.687,A -85,B 0,C 180,E1 -21050.231,E2 -21050.231} C_VEL
LIN {X 0,Y 207.06,Z 277.691,A -85,B 0,C 180,E1 -21054.156,E2 -21054.156} C_VEL
LIN {X 0,Y 207.383,Z 277.649,A -85,B 0,C 180,E1 -21058.058,E2 -21058.058} C_VEL
LIN {X 0,Y 207.506,Z 277.637,A -85,B 0,C 180,E1 -21060,E2 -21060} C_VEL
LIN {X 0,Y 207.054,Z 277.692,A -85,B 0,C 180,E1 -21063.893,E2 -21063.893} C_VEL
LIN {X 0,Y 207.136,Z 277.681,A -85,B 0,C 180,E1 -21067.8,E2 -21067.8} C_VEL
LIN {X 0,Y 206.918,Z 277.707,A -85,B 0,C 180,E1 -21071.759,E2 -21071.759} C_VEL
LIN {X 0,Y 206.844,Z 277.717,A -85,B 0,C 180,E1 -21075.773,E2 -21075.773} C_VEL
LIN {X 0,Y 206.858,Z 277.717,A -85,B 0,C 180,E1 -21077.955,E2 -21077.955} C_VEL
LIN {X 0,Y 206.755,Z 277.73,A -85,B 0,C 180,E1 -21083.396,E2 -21083.396} C_VEL
LIN {X 0,Y 206.746,Z 277.732,A -85,B 0,C 180,E1 -21088.419,E2 -21088.419} C_VEL
LIN {X 0,Y 206.71,Z 277.736,A -85,B 0,C 180,E1 -21092.956,E2 -21092.956} C_VEL
LIN {X 0,Y 206.723,Z 277.735,A -85,B 0,C 180,E1 -21095.32,E2 -21095.32} C_VEL
LIN {X 0,Y 206.664,Z 277.739,A -85,B 0,C 180,E1 -21100.251,E2 -21100.251} C_VEL
LIN {X 0,Y 206.631,Z 277.747,A -85,B 0,C 180,E1 -21105.583,E2 -21105.583} C_VEL
LIN {X 0,Y 206.946,Z 279.968,A -85,B 0,C 180,E1 -21109.816,E2 -21109.816} C_VEL
LIN {X 0,Y 207.045,Z 282.157,A -85,B 0,C 180,E1 -21113.346,E2 -21113.346} C_VEL
LIN {X 0,Y 208.125,Z 285.237,A -85,B 0,C 180,E1 -21113.763,E2 -21113.763} C_VEL
LIN {X 0,Y 210.764,Z 290.973,A -85,B 0,C 180,E1 -21114.708,E2 -21114.708} C_VEL
LIN {X 0,Y 214.269,Z 300.794,A -85,B 0,C 180,E1 -21116.287,E2 -21116.287} C_VEL
LIN {X 0,Y 217.306,Z 311.953,A -85,B 0,C 180,E1 -21118.183,E2 -21118.183} C_VEL
LIN {X 0,Y 219.149,Z 322.908,A -85,B 0,C 180,E1 -21120.173,E2 -21120.173} C_VEL
LIN {X 0,Y 220.033,Z 332.68,A -85,B 0,C 180,E1 -21122.152,E2 -21122.152} C_VEL
LIN {X 0,Y 219.875,Z 335.126,A -85,B 0,C 180,E1 -21122.647,E2 -21122.647} C_VEL
LIN {X 0,Y 217.325,Z 344.832,A -85,B 0,C 180,E1 -21124.629,E2 -21124.629} C_VEL
LIN {X 0,Y 214.835,Z 353.659,A -85,B 0,C 180,E1 -21126.886,E2 -21126.886} C_VEL
LIN {X 0,Y 212.13,Z 362.269,A -85,B 0,C 180,E1 -21129.643,E2 -21129.643} C_VEL
LIN {X 0,Y 209.71,Z 369.137,A -85,B 0,C 180,E1 -21132.445,E2 -21132.445} C_VEL
LIN {X 0,Y 207.883,Z 374.63,A -85,B 0,C 180,E1 -21135.312,E2 -21135.312} C_VEL
LIN {X 0,Y 206.442,Z 378.94,A -85,B 0,C 180,E1 -21138.214,E2 -21138.214} C_VEL
LIN {X 0,Y 205.742,Z 381.219,A -85,B 0,C 180,E1 -21140.166,E2 -21140.166} C_VEL
LIN {X 0,Y 205.202,Z 383.071,A -85,B 0,C 180,E1 -21142.126,E2 -21142.126} C_VEL
LIN {X 0,Y 204.771,Z 384.667,A -85,B 0,C 180,E1 -21144.457,E2 -21144.457} C_VEL
LIN {X 0,Y 204.496,Z 386.057,A -85,B 0,C 180,E1 -21148.031,E2 -21148.031} C_VEL
LIN {X 0,Y 204.499,Z 386.284,A -85,B 0,C 180,E1 -21150,E2 -21150} C_VEL
LIN {X 0,Y 204.496,Z 386.09,A -85,B 0,C 180,E1 -21151.97,E2 -21151.97} C_VEL
LIN {X 0,Y 204.823,Z 384.538,A -85,B 0,C 180,E1 -21155.909,E2 -21155.909} C_VEL
LIN {X 0,Y 205.204,Z 383.181,A -85,B 0,C 180,E1 -21157.874,E2 -21157.874} C_VEL
LIN {X 0,Y 206.069,Z 380.313,A -85,B 0,C 180,E1 -21160.812,E2 -21160.812} C_VEL
LIN {X 0,Y 207.317,Z 376.422,A -85,B 0,C 180,E1 -21163.727,E2 -21163.727} C_VEL
LIN {X 0,Y 209.014,Z 371.4,A -85,B 0,C 180,E1 -21166.607,E2 -21166.607} C_VEL
LIN {X 0,Y 211.2,Z 365.072,A -85,B 0,C 180,E1 -21169.437,E2 -21169.437} C_VEL
LIN {X 0,Y 213.845,Z 357.153,A -85,B 0,C 180,E1 -21172.207,E2 -21172.207} C_VEL
LIN {X 0,Y 216.375,Z 348.42,A -85,B 0,C 180,E1 -21174.656,E2 -21174.656} C_VEL
LIN {X 0,Y 219.156,Z 338.132,A -85,B 0,C 180,E1 -21176.935,E2 -21176.935} C_VEL
LIN {X 0,Y 220.062,Z 334.62,A -85,B 0,C 180,E1 -21177.586,E2 -21177.586} C_VEL
LIN {X 0,Y 219.52,Z 325.769,A -85,B 0,C 180,E1 -21179.414,E2 -21179.414} C_VEL
LIN {X 0,Y 217.895,Z 314.837,A -85,B 0,C 180,E1 -21181.47,E2 -21181.47} C_VEL
LIN {X 0,Y 215.811,Z 305.914,A -85,B 0,C 180,E1 -21183.012,E2 -21183.012} C_VEL
LIN {X 0,Y 211.908,Z 293.795,A -85,B 0,C 180,E1 -21185.002,E2 -21185.002} C_VEL
LIN {X 0,Y 208.356,Z 285.67,A -85,B 0,C 180,E1 -21186.324,E2 -21186.324} C_VEL
LIN {X 0,Y 207.134,Z 282.807,A -85,B 0,C 180,E1 -21186.765,E2 -21186.765} C_VEL
LIN {X 0,Y 207.019,Z 282.101,A -85,B 0,C 180,E1 -21186.908,E2 -21186.908} C_VEL
LIN {X 0,Y 206.947,Z 280.078,A -85,B 0,C 180,E1 -21190.185,E2 -21190.185} C_VEL
LIN {X 0,Y 206.632,Z 277.741,A -85,B 0,C 180,E1 -21194.417,E2 -21194.417} C_VEL
LIN {X 0,Y 206.665,Z 277.742,A -85,B 0,C 180,E1 -21199.749,E2 -21199.749} C_VEL
LIN {X 0,Y 206.734,Z 277.734,A -85,B 0,C 180,E1 -21204.695,E2 -21204.695} C_VEL
LIN {X 0,Y 206.726,Z 277.73,A -85,B 0,C 180,E1 -21209.339,E2 -21209.339} C_VEL
LIN {X 0,Y 206.734,Z 277.732,A -85,B 0,C 180,E1 -21213.772,E2 -21213.772} C_VEL
LIN {X 0,Y 206.738,Z 277.733,A -85,B 0,C 180,E1 -21218.041,E2 -21218.041} C_VEL
LIN {X 0,Y 206.87,Z 277.714,A -85,B 0,C 180,E1 -21222.196,E2 -21222.196} C_VEL
LIN {X 0,Y 206.887,Z 277.714,A -85,B 0,C 180,E1 -21226.244,E2 -21226.244} C_VEL
LIN {X 0,Y 207.102,Z 277.686,A -85,B 0,C 180,E1 -21230.231,E2 -21230.231} C_VEL
LIN {X 0,Y 207.048,Z 277.692,A -85,B 0,C 180,E1 -21234.155,E2 -21234.155} C_VEL
LIN {X 0,Y 207.35,Z 277.656,A -85,B 0,C 180,E1 -21238.058,E2 -21238.058} C_VEL
LIN {X 0,Y 207.485,Z 277.639,A -85,B 0,C 180,E1 -21240,E2 -21240} C_VEL
LIN {X 0,Y 207.384,Z 277.65,A -85,B 0,C 180,E1 -21241.942,E2 -21241.942} C_VEL
LIN {X 0,Y 207.14,Z 277.681,A -85,B 0,C 180,E1 -21247.8,E2 -21247.8} C_VEL
LIN {X 0,Y 206.927,Z 277.709,A -85,B 0,C 180,E1 -21251.758,E2 -21251.758} C_VEL
LIN {X 0,Y 206.87,Z 277.716,A -85,B 0,C 180,E1 -21255.77,E2 -21255.77} C_VEL
LIN {X 0,Y 206.781,Z 277.727,A -85,B 0,C 180,E1 -21259.869,E2 -21259.869} C_VEL
LIN {X 0,Y 206.734,Z 277.735,A -85,B 0,C 180,E1 -21264.076,E2 -21264.076} C_VEL
LIN {X 0,Y 206.688,Z 277.739,A -85,B 0,C 180,E1 -21268.427,E2 -21268.427} C_VEL
LIN {X 0,Y 206.696,Z 277.741,A -85,B 0,C 180,E1 -21272.958,E2 -21272.958} C_VEL
LIN {X 0,Y 206.722,Z 277.772,A -85,B 0,C 180,E1 -21275.319,E2 -21275.319} C_VEL
LIN {X 0,Y 207.063,Z 279.892,A -85,B 0,C 180,E1 -21278.679,E2 -21278.679} C_VEL
LIN {X 0,Y 207.475,Z 282.588,A -85,B 0,C 180,E1 -21282.647,E2 -21282.647} C_VEL
LIN {X 0,Y 208.064,Z 286.172,A -85,B 0,C 180,E1 -21287.502,E2 -21287.502} C_VEL
LIN {X 0,Y 208.458,Z 288.798,A -85,B 0,C 180,E1 -21290.844,E2 -21290.844} C_VEL
LIN {X 0,Y 208.489,Z 291.012,A -85,B 0,C 180,E1 -21293.491,E2 -21293.491} C_VEL
LIN {X 0,Y 209.516,Z 294.341,A -85,B 0,C 180,E1 -21293.9,E2 -21293.9} C_VEL
LIN {X 0,Y 212.232,Z 302.659,A -85,B 0,C 180,E1 -21295.029,E2 -21295.029} C_VEL
LIN {X 0,Y 215.253,Z 314.865,A -85,B 0,C 180,E1 -21296.787,E2 -21296.787} C_VEL
LIN {X 0,Y 217.059,Z 326.3,A -85,B 0,C 180,E1 -21298.596,E2 -21298.596} C_VEL
LIN {X 0,Y 217.937,Z 337.261,A -85,B 0,C 180,E1 -21300.539,E2 -21300.539} C_VEL
LIN {X 0,Y 217.911,Z 347.7,A -85,B 0,C 180,E1 -21302.639,E2 -21302.639} C_VEL
LIN {X 0,Y 217.514,Z 351.09,A -85,B 0,C 180,E1 -21303.364,E2 -21303.364} C_VEL
LIN {X 0,Y 214.379,Z 361.749,A -85,B 0,C 180,E1 -21305.808,E2 -21305.808} C_VEL
LIN {X 0,Y 212.286,Z 368.558,A -85,B 0,C 180,E1 -21307.772,E2 -21307.772} C_VEL
LIN {X 0,Y 210.548,Z 372.26,A -85,B 0,C 180,E1 -21308.941,E2 -21308.941} C_VEL
LIN {X 0,Y 206.068,Z 377.779,A -85,B 0,C 180,E1 -21310.847,E2 -21310.847} C_VEL
LIN {X 0,Y 201.672,Z 382.682,A -85,B 0,C 180,E1 -21312.941,E2 -21312.941} C_VEL
LIN {X 0,Y 200.101,Z 385.315,A -85,B 0,C 180,E1 -21314.381,E2 -21314.381} C_VEL
LIN {X 0,Y 198.605,Z 390.212,A -85,B 0,C 180,E1 -21317.741,E2 -21317.741} C_VEL
LIN {X 0,Y 198.021,Z 392.511,A -85,B 0,C 180,E1 -21319.778,E2 -21319.778} C_VEL
LIN {X 0,Y 197.579,Z 394.372,A -85,B 0,C 180,E1 -21321.82,E2 -21321.82} C_VEL
LIN {X 0,Y 197.338,Z 395.77,A -85,B 0,C 180,E1 -21323.866,E2 -21323.866} C_VEL
LIN {X 0,Y 197.25,Z 397.38,A -85,B 0,C 180,E1 -21327.958,E2 -21327.958} C_VEL
LIN {X 0,Y 197.365,Z 397.595,A -85,B 0,C 180,E1 -21330,E2 -21330} C_VEL
LIN {X 0,Y 197.204,Z 396.887,A -85,B 0,C 180,E1 -21333.739,E2 -21333.739} C_VEL
LIN {X 0,Y 197.311,Z 395.742,A -85,B 0,C 180,E1 -21336.134,E2 -21336.134} C_VEL
LIN {X 0,Y 197.568,Z 394.332,A -85,B 0,C 180,E1 -21338.18,E2 -21338.18} C_VEL
LIN {X 0,Y 198.272,Z 391.379,A -85,B 0,C 180,E1 -21341.242,E2 -21341.242} C_VEL
LIN {X 0,Y 199.386,Z 387.387,A -85,B 0,C 180,E1 -21344.284,E2 -21344.284} C_VEL
LIN {X 0,Y 201.493,Z 381.26,A -85,B 0,C 180,E1 -21347.77,E2 -21347.77} C_VEL
LIN {X 0,Y 203.795,Z 374.572,A -85,B 0,C 180,E1 -21350.7,E2 -21350.7} C_VEL
LIN {X 0,Y 206.358,Z 366.272,A -85,B 0,C 180,E1 -21353.588,E2 -21353.588} C_VEL
LIN {X 0,Y 209.04,Z 357.764,A -85,B 0,C 180,E1 -21355.917,E2 -21355.917} C_VEL
LIN {X 0,Y 211.147,Z 350.654,A -85,B 0,C 180,E1 -21357.505,E2 -21357.505} C_VEL
LIN {X 0,Y 211.453,Z 339.63,A -85,B 0,C 180,E1 -21359.904,E2 -21359.904} C_VEL
LIN {X 0,Y 210.695,Z 328.153,A -85,B 0,C 180,E1 -21362.076,E2 -21362.076} C_VEL
LIN {X 0,Y 209.283,Z 318.084,A -85,B 0,C 180,E1 -21363.785,E2 -21363.785} C_VEL
LIN {X 0,Y 206.642,Z 306.212,A -85,B 0,C 180,E1 -21365.636,E2 -21365.636} C_VEL
LIN {X 0,Y 203.917,Z 297.333,A -85,B 0,C 180,E1 -21366.965,E2 -21366.965} C_VEL
LIN {X 0,Y 202.282,Z 293.482,A -85,B 0,C 180,E1 -21367.574,E2 -21367.574} C_VEL
LIN {X 0,Y 201.463,Z 290.766,A -85,B 0,C 180,E1 -21367.93,E2 -21367.93} C_VEL
LIN {X 0,Y 201.152,Z 287.929,A -85,B 0,C 180,E1 -21371.593,E2 -21371.593} C_VEL
LIN {X 0,Y 200.641,Z 285.078,A -85,B 0,C 180,E1 -21375.528,E2 -21375.528} C_VEL
LIN {X 0,Y 200.378,Z 283.234,A -85,B 0,C 180,E1 -21378.21,E2 -21378.21} C_VEL
LIN {X 0,Y 199.924,Z 279.949,A -85,B 0,C 180,E1 -21383.301,E2 -21383.301} C_VEL
LIN {X 0,Y 199.627,Z 278.622,A -85,B 0,C 180,E1 -21385.716,E2 -21385.716} C_VEL
LIN {X 0,Y 199.686,Z 278.616,A -85,B 0,C 180,E1 -21388.134,E2 -21388.134} C_VEL
LIN {X 0,Y 199.638,Z 278.622,A -85,B 0,C 180,E1 -21392.765,E2 -21392.765} C_VEL
LIN {X 0,Y 199.706,Z 278.611,A -85,B 0,C 180,E1 -21397.225,E2 -21397.225} C_VEL
LIN {X 0,Y 199.797,Z 278.598,A -85,B 0,C 180,E1 -21401.758,E2 -21401.758} C_VEL
LIN {X 0,Y 199.837,Z 278.593,A -85,B 0,C 180,E1 -21405.748,E2 -21405.748} C_VEL
LIN {X 0,Y 200.023,Z 278.569,A -85,B 0,C 180,E1 -21409.882,E2 -21409.882} C_VEL
LIN {X 0,Y 200.021,Z 278.569,A -85,B 0,C 180,E1 -21413.949,E2 -21413.949} C_VEL
LIN {X 0,Y 200.322,Z 278.529,A -85,B 0,C 180,E1 -21417.99,E2 -21417.99} C_VEL
LIN {X 0,Y 200.471,Z 278.513,A -85,B 0,C 180,E1 -21420,E2 -21420} C_VEL
LIN {X 0,Y 200,Z 278.571,A -85,B 0,C 180,E1 -21424.03,E2 -21424.03} C_VEL
LIN {X 0,Y 200.085,Z 278.559,A -85,B 0,C 180,E1 -21428.077,E2 -21428.077} C_VEL
LIN {X 0,Y 199.868,Z 278.585,A -85,B 0,C 180,E1 -21432.18,E2 -21432.18} C_VEL
LIN {X 0,Y 199.788,Z 278.598,A -85,B 0,C 180,E1 -21436.345,E2 -21436.345} C_VEL
LIN {X 0,Y 199.675,Z 278.612,A -85,B 0,C 180,E1 -21440.608,E2 -21440.608} C_VEL
LIN {X 0,Y 199.666,Z 278.614,A -85,B 0,C 180,E1 -21444.985,E2 -21444.985} C_VEL
LIN {X 0,Y 199.676,Z 278.611,A -85,B 0,C 180,E1 -21449.522,E2 -21449.522} C_VEL
LIN {X 0,Y 199.665,Z 278.616,A -85,B 0,C 180,E1 -21452.352,E2 -21452.352} C_VEL
LIN {X 0,Y 199.64,Z 278.617,A -85,B 0,C 180,E1 -21456.76,E2 -21456.76} C_VEL
LIN {X 0,Y 199.639,Z 278.614,A -85,B 0,C 180,E1 -21459.321,E2 -21459.321} C_VEL
LIN {X 0,Y 199.577,Z 278.623,A -85,B 0,C 180,E1 -21464.772,E2 -21464.772} C_VEL
LIN {X 0,Y 199.836,Z 280.205,A -85,B 0,C 180,E1 -21468.071,E2 -21468.071} C_VEL
LIN {X 0,Y 200.094,Z 282.457,A -85,B 0,C 180,E1 -21471.851,E2 -21471.851} C_VEL
LIN {X 0,Y 201.273,Z 285.627,A -85,B 0,C 180,E1 -21472.329,E2 -21472.329} C_VEL
LIN {X 0,Y 205.373,Z 294.624,A -85,B 0,C 180,E1 -21473.937,E2 -21473.937} C_VEL
LIN {X 0,Y 208.928,Z 305.403,A -85,B 0,C 180,E1 -21475.819,E2 -21475.819} C_VEL
LIN {X 0,Y 211.273,Z 314.764,A -85,B 0,C 180,E1 -21477.537,E2 -21477.537} C_VEL
LIN {X 0,Y 212.881,Z 325.583,A -85,B 0,C 180,E1 -21479.649,E2 -21479.649} C_VEL
LIN {X 0,Y 213.567,Z 335.331,A -85,B 0,C 180,E1 -21481.768,E2 -21481.768} C_VEL
LIN {X 0,Y 210.937,Z 345.034,A -85,B 0,C 180,E1 -21483.803,E2 -21483.803} C_VEL
LIN {X 0,Y 208.311,Z 353.862,A -85,B 0,C 180,E1 -21486.118,E2 -21486.118} C_VEL
LIN {X 0,Y 205.488,Z 362.471,A -85,B 0,C 180,E1 -21488.954,E2 -21488.954} C_VEL
LIN {X 0,Y 202.941,Z 369.339,A -85,B 0,C 180,E1 -21491.84,E2 -21491.84} C_VEL
LIN {X 0,Y 201.015,Z 374.831,A -85,B 0,C 180,E1 -21494.798,E2 -21494.798} C_VEL
LIN {X 0,Y 199.496,Z 379.141,A -85,B 0,C 180,E1 -21497.797,E2 -21497.797} C_VEL
LIN {X 0,Y 198.755,Z 381.419,A -85,B 0,C 180,E1 -21499.817,E2 -21499.817} C_VEL
LIN {X 0,Y 198.165,Z 383.271,A -85,B 0,C 180,E1 -21501.845,E2 -21501.845} C_VEL
LIN {X 0,Y 197.64,Z 385.092,A -85,B 0,C 180,E1 -21504.669,E2 -21504.669} C_VEL
LIN {X 0,Y 197.403,Z 386.257,A -85,B 0,C 180,E1 -21507.96,E2 -21507.96} C_VEL
LIN {X 0,Y 197.401,Z 386.483,A -85,B 0,C 180,E1 -21510,E2 -21510} C_VEL
LIN {X 0,Y 197.403,Z 386.29,A -85,B 0,C 180,E1 -21512.041,E2 -21512.041} C_VEL
LIN {X 0,Y 197.766,Z 384.738,A -85,B 0,C 180,E1 -21516.12,E2 -21516.12} C_VEL
LIN {X 0,Y 198.166,Z 383.381,A -85,B 0,C 180,E1 -21518.156,E2 -21518.156} C_VEL
LIN {X 0,Y 199.102,Z 380.512,A -85,B 0,C 180,E1 -21521.195,E2 -21521.195} C_VEL
LIN {X 0,Y 200.43,Z 376.621,A -85,B 0,C 180,E1 -21524.209,E2 -21524.209} C_VEL
LIN {X 0,Y 202.211,Z 371.599,A -85,B 0,C 180,E1 -21527.183,E2 -21527.183} C_VEL
LIN {X 0,Y 204.516,Z 365.27,A -85,B 0,C 180,E1 -21530.099,E2 -21530.099} C_VEL
LIN {X 0,Y 207.284,Z 357.35,A -85,B 0,C 180,E1 -21532.949,E2 -21532.949} C_VEL
LIN {X 0,Y 209.866,Z 348.864,A -85,B 0,C 180,E1 -21535.4,E2 -21535.4} C_VEL
LIN {X 0,Y 212.549,Z 339.428,A -85,B 0,C 180,E1 -21537.576,E2 -21537.576} C_VEL
LIN {X 0,Y 213.584,Z 334.823,A -85,B 0,C 180,E1 -21538.498,E2 -21538.498} C_VEL
LIN {X 0,Y 212.947,Z 325.678,A -85,B 0,C 180,E1 -21540.475,E2 -21540.475} C_VEL
LIN {X 0,Y 211.224,Z 314.354,A -85,B 0,C 180,E1 -21542.689,E2 -21542.689} C_VEL
LIN {X 0,Y 208.472,Z 303.847,A -85,B 0,C 180,E1 -21544.621,E2 -21544.621} C_VEL
LIN {X 0,Y 204.973,Z 293.682,A -85,B 0,C 180,E1 -21546.402,E2 -21546.402} C_VEL
LIN {X 0,Y 201.359,Z 285.791,A -85,B 0,C 180,E1 -21547.81,E2 -21547.81} C_VEL
LIN {X 0,Y 200.108,Z 282.661,A -85,B 0,C 180,E1 -21548.305,E2 -21548.305} C_VEL
LIN {X 0,Y 200.063,Z 282.362,A -85,B 0,C 180,E1 -21548.39,E2 -21548.39} C_VEL
LIN {X 0,Y 199.806,Z 280.061,A -85,B 0,C 180,E1 -21552.383,E2 -21552.383} C_VEL
LIN {X 0,Y 199.578,Z 278.621,A -85,B 0,C 180,E1 -21555.228,E2 -21555.228} C_VEL
LIN {X 0,Y 199.64,Z 278.616,A -85,B 0,C 180,E1 -21560.679,E2 -21560.679} C_VEL
LIN {X 0,Y 199.637,Z 278.616,A -85,B 0,C 180,E1 -21565.718,E2 -21565.718} C_VEL
LIN {X 0,Y 199.706,Z 278.607,A -85,B 0,C 180,E1 -21568.138,E2 -21568.138} C_VEL
LIN {X 0,Y 199.689,Z 278.606,A -85,B 0,C 180,E1 -21572.772,E2 -21572.772} C_VEL
LIN {X 0,Y 199.715,Z 278.601,A -85,B 0,C 180,E1 -21577.226,E2 -21577.226} C_VEL
LIN {X 0,Y 199.797,Z 278.597,A -85,B 0,C 180,E1 -21581.759,E2 -21581.759} C_VEL
LIN {X 0,Y 199.825,Z 278.594,A -85,B 0,C 180,E1 -21585.747,E2 -21585.747} C_VEL
LIN {X 0,Y 200.025,Z 278.568,A -85,B 0,C 180,E1 -21589.882,E2 -21589.882} C_VEL
LIN {X 0,Y 200.011,Z 278.569,A -85,B 0,C 180,E1 -21593.949,E2 -21593.949} C_VEL
LIN {X 0,Y 200.292,Z 278.535,A -85,B 0,C 180,E1 -21597.989,E2 -21597.989} C_VEL
LIN {X 0,Y 200.452,Z 278.515,A -85,B 0,C 180,E1 -21600,E2 -21600} C_VEL
LIN {X 0,Y 200.323,Z 278.53,A -85,B 0,C 180,E1 -21602.01,E2 -21602.01} C_VEL
LIN {X 0,Y 200.089,Z 278.56,A -85,B 0,C 180,E1 -21608.077,E2 -21608.077} C_VEL
LIN {X 0,Y 199.877,Z 278.587,A -85,B 0,C 180,E1 -21612.179,E2 -21612.179} C_VEL
LIN {X 0,Y 199.807,Z 278.597,A -85,B 0,C 180,E1 -21616.343,E2 -21616.343} C_VEL
LIN {X 0,Y 199.692,Z 278.61,A -85,B 0,C 180,E1 -21620.606,E2 -21620.606} C_VEL
LIN {X 0,Y 199.646,Z 278.616,A -85,B 0,C 180,E1 -21624.988,E2 -21624.988} C_VEL
LIN {X 0,Y 199.609,Z 278.622,A -85,B 0,C 180,E1 -21629.533,E2 -21629.533} C_VEL
LIN {X 0,Y 199.648,Z 278.618,A -85,B 0,C 180,E1 -21632.344,E2 -21632.344} C_VEL
LIN {X 0,Y 199.721,Z 278.841,A -85,B 0,C 180,E1 -21634.702,E2 -21634.702} C_VEL
LIN {X 0,Y 200.137,Z 281.742,A -85,B 0,C 180,E1 -21639.416,E2 -21639.416} C_VEL
LIN {X 0,Y 200.5,Z 283.834,A -85,B 0,C 180,E1 -21642.599,E2 -21642.599} C_VEL
LIN {X 0,Y 201.035,Z 287.127,A -85,B 0,C 180,E1 -21647.235,E2 -21647.235} C_VEL
LIN {X 0,Y 201.438,Z 290.065,A -85,B 0,C 180,E1 -21651.096,E2 -21651.096} C_VEL
LIN {X 0,Y 201.478,Z 290.771,A -85,B 0,C 180,E1 -21651.986,E2 -21651.986} C_VEL
LIN {X 0,Y 202.599,Z 294.155,A -85,B 0,C 180,E1 -21652.463,E2 -21652.463} C_VEL
LIN {X 0,Y 204.624,Z 299.15,A -85,B 0,C 180,E1 -21653.253,E2 -21653.253} C_VEL
LIN {X 0,Y 207.653,Z 309.993,A -85,B 0,C 180,E1 -21654.875,E2 -21654.875} C_VEL
LIN {X 0,Y 209.785,Z 320.789,A -85,B 0,C 180,E1 -21656.599,E2 -21656.599} C_VEL
LIN {X 0,Y 211.033,Z 331.212,A -85,B 0,C 180,E1 -21658.42,E2 -21658.42} C_VEL
LIN {X 0,Y 211.466,Z 341.289,A -85,B 0,C 180,E1 -21660.379,E2 -21660.379} C_VEL
LIN {X 0,Y 211.166,Z 350.892,A -85,B 0,C 180,E1 -21662.497,E2 -21662.497} C_VEL
LIN {X 0,Y 207.893,Z 361.551,A -85,B 0,C 180,E1 -21665.003,E2 -21665.003} C_VEL
LIN {X 0,Y 204.967,Z 370.65,A -85,B 0,C 180,E1 -21667.788,E2 -21667.788} C_VEL
LIN {X 0,Y 202.911,Z 377.096,A -85,B 0,C 180,E1 -21670.263,E2 -21670.263} C_VEL
LIN {X 0,Y 201.137,Z 382.363,A -85,B 0,C 180,E1 -21672.722,E2 -21672.722} C_VEL
LIN {X 0,Y 200.101,Z 385.315,A -85,B 0,C 180,E1 -21674.381,E2 -21674.381} C_VEL
LIN {X 0,Y 198.635,Z 387.754,A -85,B 0,C 180,E1 -21675.875,E2 -21675.875} C_VEL
LIN {X 0,Y 194.784,Z 391.121,A -85,B 0,C 180,E1 -21678.355,E2 -21678.355} C_VEL
LIN {X 0,Y 191.826,Z 393.261,A -85,B 0,C 180,E1 -21680.451,E2 -21680.451} C_VEL
LIN {X 0,Y 190.507,Z 394.606,A -85,B 0,C 180,E1 -21682.136,E2 -21682.136} C_VEL
LIN {X 0,Y 190.354,Z 394.964,A -85,B 0,C 180,E1 -21682.716,E2 -21682.716} C_VEL
LIN {X 0,Y 190.101,Z 396.864,A -85,B 0,C 180,E1 -21686.549,E2 -21686.549} C_VEL
LIN {X 0,Y 190.267,Z 397.395,A -85,B 0,C 180,E1 -21690,E2 -21690} C_VEL
LIN {X 0,Y 190.122,Z 396.812,A -85,B 0,C 180,E1 -21693.552,E2 -21693.552} C_VEL
LIN {X 0,Y 190.231,Z 395.541,A -85,B 0,C 180,E1 -21696.363,E2 -21696.363} C_VEL
LIN {X 0,Y 190.522,Z 394.131,A -85,B 0,C 180,E1 -21698.485,E2 -21698.485} C_VEL
LIN {X 0,Y 191.284,Z 391.178,A -85,B 0,C 180,E1 -21701.658,E2 -21701.658} C_VEL
LIN {X 0,Y 192.473,Z 387.185,A -85,B 0,C 180,E1 -21704.809,E2 -21704.809} C_VEL
LIN {X 0,Y 194.726,Z 381.058,A -85,B 0,C 180,E1 -21708.409,E2 -21708.409} C_VEL
LIN {X 0,Y 197.116,Z 374.482,A -85,B 0,C 180,E1 -21711.386,E2 -21711.386} C_VEL
LIN {X 0,Y 199.837,Z 366.069,A -85,B 0,C 180,E1 -21714.407,E2 -21714.407} C_VEL
LIN {X 0,Y 202.664,Z 357.561,A -85,B 0,C 180,E1 -21716.796,E2 -21716.796} C_VEL
LIN {X 0,Y 204.544,Z 351.523,A -85,B 0,C 180,E1 -21718.193,E2 -21718.193} C_VEL
LIN {X 0,Y 204.956,Z 340.929,A -85,B 0,C 180,E1 -21720.629,E2 -21720.629} C_VEL
LIN {X 0,Y 204.489,Z 331.078,A -85,B 0,C 180,E1 -21722.632,E2 -21722.632} C_VEL
LIN {X 0,Y 203.128,Z 319.676,A -85,B 0,C 180,E1 -21724.709,E2 -21724.709} C_VEL
LIN {X 0,Y 200.518,Z 307.428,A -85,B 0,C 180,E1 -21726.754,E2 -21726.754} C_VEL
LIN {X 0,Y 197.825,Z 298.834,A -85,B 0,C 180,E1 -21728.158,E2 -21728.158} C_VEL
LIN {X 0,Y 195.847,Z 294.391,A -85,B 0,C 180,E1 -21728.953,E2 -21728.953} C_VEL
LIN {X 0,Y 194.573,Z 291.512,A -85,B 0,C 180,E1 -21729.46,E2 -21729.46} C_VEL
LIN {X 0,Y 194.375,Z 290.51,A -85,B 0,C 180,E1 -21729.593,E2 -21729.593} C_VEL
LIN {X 0,Y 193.903,Z 287.671,A -85,B 0,C 180,E1 -21733.54,E2 -21733.54} C_VEL
LIN {X 0,Y 193.548,Z 285.6,A -85,B 0,C 180,E1 -21736.571,E2 -21736.571} C_VEL
LIN {X 0,Y 193.048,Z 282.281,A -85,B 0,C 180,E1 -21741.765,E2 -21741.765} C_VEL
LIN {X 0,Y 192.705,Z 280.073,A -85,B 0,C 180,E1 -21745.578,E2 -21745.578} C_VEL
LIN {X 0,Y 192.6,Z 279.499,A -85,B 0,C 180,E1 -21747.064,E2 -21747.064} C_VEL
LIN {X 0,Y 192.619,Z 279.497,A -85,B 0,C 180,E1 -21751.685,E2 -21751.685} C_VEL
LIN {X 0,Y 192.675,Z 279.487,A -85,B 0,C 180,E1 -21756.345,E2 -21756.345} C_VEL
LIN {X 0,Y 192.732,Z 279.478,A -85,B 0,C 180,E1 -21761.458,E2 -21761.458} C_VEL
LIN {X 0,Y 192.765,Z 279.473,A -85,B 0,C 180,E1 -21765.214,E2 -21765.214} C_VEL
LIN {X 0,Y 192.946,Z 279.449,A -85,B 0,C 180,E1 -21769.567,E2 -21769.567} C_VEL
LIN {X 0,Y 192.984,Z 279.447,A -85,B 0,C 180,E1 -21773.728,E2 -21773.728} C_VEL
LIN {X 0,Y 193.264,Z 279.408,A -85,B 0,C 180,E1 -21777.916,E2 -21777.916} C_VEL
LIN {X 0,Y 193.434,Z 279.39,A -85,B 0,C 180,E1 -21780,E2 -21780} C_VEL
LIN {X 0,Y 192.948,Z 279.449,A -85,B 0,C 180,E1 -21784.178,E2 -21784.178} C_VEL
LIN {X 0,Y 193.034,Z 279.437,A -85,B 0,C 180,E1 -21788.374,E2 -21788.374} C_VEL
LIN {X 0,Y 192.795,Z 279.468,A -85,B 0,C 180,E1 -21792.634,E2 -21792.634} C_VEL
LIN {X 0,Y 192.747,Z 279.476,A -85,B 0,C 180,E1 -21796.96,E2 -21796.96} C_VEL
LIN {X 0,Y 192.612,Z 279.49,A -85,B 0,C 180,E1 -21801.4,E2 -21801.4} C_VEL
LIN {X 0,Y 192.648,Z 279.487,A -85,B 0,C 180,E1 -21804.213,E2 -21804.213} C_VEL
LIN {X 0,Y 192.651,Z 279.486,A -85,B 0,C 180,E1 -21808.892,E2 -21808.892} C_VEL
LIN {X 0,Y 192.602,Z 279.494,A -85,B 0,C 180,E1 -21813.186,E2 -21813.186} C_VEL
LIN {X 0,Y 192.61,Z 279.493,A -85,B 0,C 180,E1 -21816.607,E2 -21816.607} C_VEL
LIN {X 0,Y 192.521,Z 279.505,A -85,B 0,C 180,E1 -21821.079,E2 -21821.079} C_VEL
LIN {X 0,Y 192.49,Z 279.509,A -85,B 0,C 180,E1 -21823.925,E2 -21823.925} C_VEL
LIN {X 0,Y 192.731,Z 280.82,A -85,B 0,C 180,E1 -21826.829,E2 -21826.829} C_VEL
LIN {X 0,Y 192.966,Z 282.619,A -85,B 0,C 180,E1 -21830.159,E2 -21830.159} C_VEL
LIN {X 0,Y 194.259,Z 285.862,A -85,B 0,C 180,E1 -21830.711,E2 -21830.711} C_VEL
LIN {X 0,Y 195.385,Z 287.767,A -85,B 0,C 180,E1 -21831.123,E2 -21831.123} C_VEL
LIN {X 0,Y 199.971,Z 298.38,A -85,B 0,C 180,E1 -21833.172,E2 -21833.172} C_VEL
LIN {X 0,Y 203.185,Z 308.787,A -85,B 0,C 180,E1 -21835.141,E2 -21835.141} C_VEL
LIN {X 0,Y 205.309,Z 318.134,A -85,B 0,C 180,E1 -21836.999,E2 -21836.999} C_VEL
LIN {X 0,Y 206.699,Z 329.239,A -85,B 0,C 180,E1 -21839.335,E2 -21839.335} C_VEL
LIN {X 0,Y 207.032,Z 336.703,A -85,B 0,C 180,E1 -21841.07,E2 -21841.07} C_VEL
LIN {X 0,Y 204.024,Z 347.18,A -85,B 0,C 180,E1 -21843.397,E2 -21843.397} C_VEL
LIN {X 0,Y 201.331,Z 355.657,A -85,B 0,C 180,E1 -21845.785,E2 -21845.785} C_VEL
LIN {X 0,Y 198.423,Z 363.9,A -85,B 0,C 180,E1 -21848.713,E2 -21848.713} C_VEL
LIN {X 0,Y 196.2,Z 369.541,A -85,B 0,C 180,E1 -21851.193,E2 -21851.193} C_VEL
LIN {X 0,Y 194.171,Z 375.033,A -85,B 0,C 180,E1 -21854.249,E2 -21854.249} C_VEL
LIN {X 0,Y 192.57,Z 379.342,A -85,B 0,C 180,E1 -21857.351,E2 -21857.351} C_VEL
LIN {X 0,Y 191.765,Z 381.62,A -85,B 0,C 180,E1 -21859.441,E2 -21859.441} C_VEL
LIN {X 0,Y 191.128,Z 383.472,A -85,B 0,C 180,E1 -21861.542,E2 -21861.542} C_VEL
LIN {X 0,Y 190.529,Z 385.486,A -85,B 0,C 180,E1 -21864.841,E2 -21864.841} C_VEL
LIN {X 0,Y 190.313,Z 386.457,A -85,B 0,C 180,E1 -21867.884,E2 -21867.884} C_VEL
LIN {X 0,Y 190.305,Z 386.683,A -85,B 0,C 180,E1 -21870,E2 -21870} C_VEL
LIN {X 0,Y 190.312,Z 386.49,A -85,B 0,C 180,E1 -21872.117,E2 -21872.117} C_VEL
LIN {X 0,Y 190.537,Z 385.542,A -85,B 0,C 180,E1 -21875.185,E2 -21875.185} C_VEL
LIN {X 0,Y 191.129,Z 383.58,A -85,B 0,C 180,E1 -21878.458,E2 -21878.458} C_VEL
LIN {X 0,Y 192.131,Z 380.711,A -85,B 0,C 180,E1 -21881.607,E2 -21881.607} C_VEL
LIN {X 0,Y 193.547,Z 376.819,A -85,B 0,C 180,E1 -21884.725,E2 -21884.725} C_VEL
LIN {X 0,Y 195.435,Z 371.797,A -85,B 0,C 180,E1 -21887.799,E2 -21887.799} C_VEL
LIN {X 0,Y 197.855,Z 365.468,A -85,B 0,C 180,E1 -21890.807,E2 -21890.807} C_VEL
LIN {X 0,Y 200.76,Z 357.548,A -85,B 0,C 180,E1 -21893.74,E2 -21893.74} C_VEL
LIN {X 0,Y 203.364,Z 349.368,A -85,B 0,C 180,E1 -21896.178,E2 -21896.178} C_VEL
LIN {X 0,Y 206.293,Z 339.624,A -85,B 0,C 180,E1 -21898.487,E2 -21898.487} C_VEL
LIN {X 0,Y 207.072,Z 336.188,A -85,B 0,C 180,E1 -21899.202,E2 -21899.202} C_VEL
LIN {X 0,Y 206.493,Z 326.793,A -85,B 0,C 180,E1 -21901.35,E2 -21901.35} C_VEL
LIN {X 0,Y 205.18,Z 317.165,A -85,B 0,C 180,E1 -21903.349,E2 -21903.349} C_VEL
LIN {X 0,Y 202.641,Z 306.759,A -85,B 0,C 180,E1 -21905.409,E2 -21905.409} C_VEL
LIN {X 0,Y 199.497,Z 297.231,A -85,B 0,C 180,E1 -21907.222,E2 -21907.222} C_VEL
LIN {X 0,Y 195.102,Z 287.016,A -85,B 0,C 180,E1 -21909.175,E2 -21909.175} C_VEL
LIN {X 0,Y 193.35,Z 284.107,A -85,B 0,C 180,E1 -21909.821,E2 -21909.821} C_VEL
LIN {X 0,Y 192.956,Z 282.579,A -85,B 0,C 180,E1 -21910.103,E2 -21910.103} C_VEL
LIN {X 0,Y 192.656,Z 280.554,A -85,B 0,C 180,E1 -21913.877,E2 -21913.877} C_VEL
LIN {X 0,Y 192.491,Z 279.505,A -85,B 0,C 180,E1 -21916.076,E2 -21916.076} C_VEL
LIN {X 0,Y 192.541,Z 279.503,A -85,B 0,C 180,E1 -21920.043,E2 -21920.043} C_VEL
LIN {X 0,Y 192.601,Z 279.495,A -85,B 0,C 180,E1 -21924.279,E2 -21924.279} C_VEL
LIN {X 0,Y 192.61,Z 279.488,A -85,B 0,C 180,E1 -21929.28,E2 -21929.28} C_VEL
LIN {X 0,Y 192.667,Z 279.483,A -85,B 0,C 180,E1 -21931.692,E2 -21931.692} C_VEL
LIN {X 0,Y 192.687,Z 279.476,A -85,B 0,C 180,E1 -21936.346,E2 -21936.346} C_VEL
LIN {X 0,Y 192.732,Z 279.479,A -85,B 0,C 180,E1 -21941.46,E2 -21941.46} C_VEL
LIN {X 0,Y 192.754,Z 279.474,A -85,B 0,C 180,E1 -21945.213,E2 -21945.213} C_VEL
LIN {X 0,Y 192.947,Z 279.451,A -85,B 0,C 180,E1 -21949.567,E2 -21949.567} C_VEL
LIN {X 0,Y 192.975,Z 279.446,A -85,B 0,C 180,E1 -21953.727,E2 -21953.727} C_VEL
LIN {X 0,Y 193.237,Z 279.414,A -85,B 0,C 180,E1 -21957.916,E2 -21957.916} C_VEL
LIN {X 0,Y 193.418,Z 279.391,A -85,B 0,C 180,E1 -21960,E2 -21960} C_VEL
LIN {X 0,Y 192.975,Z 279.448,A -85,B 0,C 180,E1 -21964.177,E2 -21964.177} C_VEL
LIN {X 0,Y 193.037,Z 279.44,A -85,B 0,C 180,E1 -21968.374,E2 -21968.374} C_VEL
LIN {X 0,Y 192.805,Z 279.468,A -85,B 0,C 180,E1 -21972.633,E2 -21972.633} C_VEL
LIN {X 0,Y 192.76,Z 279.472,A -85,B 0,C 180,E1 -21976.958,E2 -21976.958} C_VEL
LIN {X 0,Y 192.62,Z 279.491,A -85,B 0,C 180,E1 -21981.399,E2 -21981.399} C_VEL
LIN {X 0,Y 192.637,Z 279.491,A -85,B 0,C 180,E1 -21984.205,E2 -21984.205} C_VEL
LIN {X 0,Y 192.602,Z 279.494,A -85,B 0,C 180,E1 -21988.865,E2 -21988.865} C_VEL
LIN {X 0,Y 192.638,Z 279.627,A -85,B 0,C 180,E1 -21993.491,E2 -21993.491} C_VEL
LIN {X 0,Y 193.055,Z 282.35,A -85,B 0,C 180,E1 -21998.234,E2 -21998.234} C_VEL
LIN {X 0,Y 193.599,Z 285.776,A -85,B 0,C 180,E1 -22003.609,E2 -22003.609} C_VEL
LIN {X 0,Y 194.102,Z 288.79,A -85,B 0,C 180,E1 -22007.945,E2 -22007.945} C_VEL
LIN {X 0,Y 194.378,Z 290.6,A -85,B 0,C 180,E1 -22010.355,E2 -22010.355} C_VEL
LIN {X 0,Y 195.345,Z 293.544,A -85,B 0,C 180,E1 -22010.783,E2 -22010.783} C_VEL
LIN {X 0,Y 196.665,Z 296.103,A -85,B 0,C 180,E1 -22011.276,E2 -22011.276} C_VEL
LIN {X 0,Y 199.361,Z 303.197,A -85,B 0,C 180,E1 -22012.486,E2 -22012.486} C_VEL
LIN {X 0,Y 202.165,Z 314.31,A -85,B 0,C 180,E1 -22014.307,E2 -22014.307} C_VEL
LIN {X 0,Y 204.05,Z 325.877,A -85,B 0,C 180,E1 -22016.338,E2 -22016.338} C_VEL
LIN {X 0,Y 204.859,Z 336.206,A -85,B 0,C 180,E1 -22018.323,E2 -22018.323} C_VEL
LIN {X 0,Y 204.916,Z 346.562,A -85,B 0,C 180,E1 -22020.569,E2 -22020.569} C_VEL
LIN {X 0,Y 204.557,Z 351.767,A -85,B 0,C 180,E1 -22021.809,E2 -22021.809} C_VEL
LIN {X 0,Y 201.469,Z 361.354,A -85,B 0,C 180,E1 -22024.148,E2 -22024.148} C_VEL
LIN {X 0,Y 198.804,Z 369.214,A -85,B 0,C 180,E1 -22026.565,E2 -22026.565} C_VEL
LIN {X 0,Y 196.227,Z 376.897,A -85,B 0,C 180,E1 -22029.561,E2 -22029.561} C_VEL
LIN {X 0,Y 194.353,Z 382.164,A -85,B 0,C 180,E1 -22032.099,E2 -22032.099} C_VEL
LIN {X 0,Y 192.475,Z 387.266,A -85,B 0,C 180,E1 -22035.191,E2 -22035.191} C_VEL
LIN {X 0,Y 191.284,Z 391.236,A -85,B 0,C 180,E1 -22038.341,E2 -22038.341} C_VEL
LIN {X 0,Y 190.53,Z 394.172,A -85,B 0,C 180,E1 -22041.515,E2 -22041.515} C_VEL
LIN {X 0,Y 190.354,Z 394.964,A -85,B 0,C 180,E1 -22042.716,E2 -22042.716} C_VEL
LIN {X 0,Y 189.539,Z 396.001,A -85,B 0,C 180,E1 -22044.454,E2 -22044.454} C_VEL
LIN {X 0,Y 187.882,Z 396.687,A -85,B 0,C 180,E1 -22046.174,E2 -22046.174} C_VEL
LIN {X 0,Y 184.151,Z 397.209,A -85,B 0,C 180,E1 -22049.685,E2 -22049.685} C_VEL
LIN {X 0,Y 183.13,Z 397.086,A -85,B 0,C 180,E1 -22051.525,E2 -22051.525} C_VEL
LIN {X 0,Y 183.052,Z 396.973,A -85,B 0,C 180,E1 -22052.149,E2 -22052.149} C_VEL
LIN {X 0,Y 183.035,Z 396.348,A -85,B 0,C 180,E1 -22054.404,E2 -22054.404} C_VEL
LIN {X 0,Y 183.178,Z 395.341,A -85,B 0,C 180,E1 -22056.609,E2 -22056.609} C_VEL
LIN {X 0,Y 183.495,Z 393.931,A -85,B 0,C 180,E1 -22058.812,E2 -22058.812} C_VEL
LIN {X 0,Y 184.317,Z 390.976,A -85,B 0,C 180,E1 -22062.105,E2 -22062.105} C_VEL
LIN {X 0,Y 185.58,Z 386.983,A -85,B 0,C 180,E1 -22065.372,E2 -22065.372} C_VEL
LIN {X 0,Y 187.98,Z 380.856,A -85,B 0,C 180,E1 -22069.095,E2 -22069.095} C_VEL
LIN {X 0,Y 190.675,Z 373.736,A -85,B 0,C 180,E1 -22072.396,E2 -22072.396} C_VEL
LIN {X 0,Y 193.357,Z 365.864,A -85,B 0,C 180,E1 -22075.282,E2 -22075.282} C_VEL
LIN {X 0,Y 196.348,Z 357.358,A -85,B 0,C 180,E1 -22077.731,E2 -22077.731} C_VEL
LIN {X 0,Y 197.976,Z 352.392,A -85,B 0,C 180,E1 -22078.926,E2 -22078.926} C_VEL
LIN {X 0,Y 198.508,Z 341.881,A -85,B 0,C 180,E1 -22081.471,E2 -22081.471} C_VEL
LIN {X 0,Y 198.126,Z 331.763,A -85,B 0,C 180,E1 -22083.645,E2 -22083.645} C_VEL
LIN {X 0,Y 196.858,Z 320.559,A -85,B 0,C 180,E1 -22085.81,E2 -22085.81} C_VEL
LIN {X 0,Y 194.472,Z 308.887,A -85,B 0,C 180,E1 -22087.905,E2 -22087.905} C_VEL
LIN {X 0,Y 192.177,Z 301.709,A -85,B 0,C 180,E1 -22089.209,E2 -22089.209} C_VEL
LIN {X 0,Y 189.014,Z 294.639,A -85,B 0,C 180,E1 -22090.609,E2 -22090.609} C_VEL
LIN {X 0,Y 187.473,Z 291.716,A -85,B 0,C 180,E1 -22091.236,E2 -22091.236} C_VEL
LIN {X 0,Y 187.12,Z 290.237,A -85,B 0,C 180,E1 -22091.499,E2 -22091.499} C_VEL
LIN {X 0,Y 186.607,Z 287.41,A -85,B 0,C 180,E1 -22095.691,E2 -22095.691} C_VEL
LIN {X 0,Y 186.226,Z 284.645,A -85,B 0,C 180,E1 -22100.091,E2 -22100.091} C_VEL
LIN {X 0,Y 186.009,Z 283.037,A -85,B 0,C 180,E1 -22102.805,E2 -22102.805} C_VEL
LIN {X 0,Y 185.556,Z 280.48,A -85,B 0,C 180,E1 -22107.578,E2 -22107.578} C_VEL
LIN {X 0,Y 185.547,Z 280.378,A -85,B 0,C 180,E1 -22110.595,E2 -22110.595} C_VEL
LIN {X 0,Y 185.581,Z 280.373,A -85,B 0,C 180,E1 -22115.382,E2 -22115.382} C_VEL
LIN {X 0,Y 185.675,Z 280.357,A -85,B 0,C 180,E1 -22121.134,E2 -22121.134} C_VEL
LIN {X 0,Y 185.696,Z 280.353,A -85,B 0,C 180,E1 -22124.637,E2 -22124.637} C_VEL
LIN {X 0,Y 185.889,Z 280.328,A -85,B 0,C 180,E1 -22129.418,E2 -22129.418} C_VEL
LIN {X 0,Y 185.947,Z 280.324,A -85,B 0,C 180,E1 -22133.489,E2 -22133.489} C_VEL
LIN {X 0,Y 186.208,Z 280.287,A -85,B 0,C 180,E1 -22137.837,E2 -22137.837} C_VEL
LIN {X 0,Y 186.398,Z 280.266,A -85,B 0,C 180,E1 -22140,E2 -22140} C_VEL
LIN {X 0,Y 185.896,Z 280.328,A -85,B 0,C 180,E1 -22144.337,E2 -22144.337} C_VEL
LIN {X 0,Y 185.981,Z 280.316,A -85,B 0,C 180,E1 -22148.694,E2 -22148.694} C_VEL
LIN {X 0,Y 185.722,Z 280.352,A -85,B 0,C 180,E1 -22153.124,E2 -22153.124} C_VEL
LIN {X 0,Y 185.684,Z 280.354,A -85,B 0,C 180,E1 -22157.626,E2 -22157.626} C_VEL
LIN {X 0,Y 185.576,Z 280.368,A -85,B 0,C 180,E1 -22162.254,E2 -22162.254} C_VEL
LIN {X 0,Y 185.562,Z 280.37,A -85,B 0,C 180,E1 -22167.032,E2 -22167.032} C_VEL
LIN {X 0,Y 185.58,Z 280.366,A -85,B 0,C 180,E1 -22169.493,E2 -22169.493} C_VEL
LIN {X 0,Y 185.52,Z 280.377,A -85,B 0,C 180,E1 -22174.628,E2 -22174.628} C_VEL
LIN {X 0,Y 185.545,Z 280.372,A -85,B 0,C 180,E1 -22177.304,E2 -22177.304} C_VEL
LIN {X 0,Y 185.484,Z 280.379,A -85,B 0,C 180,E1 -22180.729,E2 -22180.729} C_VEL
LIN {X 0,Y 185.457,Z 280.381,A -85,B 0,C 180,E1 -22183.01,E2 -22183.01} C_VEL
LIN {X 0,Y 185.818,Z 282.71,A -85,B 0,C 180,E1 -22187.982,E2 -22187.982} C_VEL
LIN {X 0,Y 185.876,Z 283.082,A -85,B 0,C 180,E1 -22188.325,E2 -22188.325} C_VEL
LIN {X 0,Y 187.2,Z 286.237,A -85,B 0,C 180,E1 -22188.928,E2 -22188.928} C_VEL
LIN {X 0,Y 188.627,Z 288.486,A -85,B 0,C 180,E1 -22189.483,E2 -22189.483} C_VEL
LIN {X 0,Y 192.162,Z 295.981,A -85,B 0,C 180,E1 -22191.109,E2 -22191.109} C_VEL
LIN {X 0,Y 195.764,Z 305.729,A -85,B 0,C 180,E1 -22193.139,E2 -22193.139} C_VEL
LIN {X 0,Y 198.742,Z 318.051,A -85,B 0,C 180,E1 -22195.706,E2 -22195.706} C_VEL
LIN {X 0,Y 200.068,Z 327.943,A -85,B 0,C 180,E1 -22197.883,E2 -22197.883} C_VEL
LIN {X 0,Y 200.541,Z 338.076,A -85,B 0,C 180,E1 -22200.329,E2 -22200.329} C_VEL
LIN {X 0,Y 197.691,Z 347.384,A -85,B 0,C 180,E1 -22202.474,E2 -22202.474} C_VEL
LIN {X 0,Y 194.872,Z 355.859,A -85,B 0,C 180,E1 -22204.928,E2 -22204.928} C_VEL
LIN {X 0,Y 191.82,Z 364.102,A -85,B 0,C 180,E1 -22207.942,E2 -22207.942} C_VEL
LIN {X 0,Y 189.492,Z 369.742,A -85,B 0,C 180,E1 -22210.501,E2 -22210.501} C_VEL
LIN {X 0,Y 187.331,Z 375.234,A -85,B 0,C 180,E1 -22213.658,E2 -22213.658} C_VEL
LIN {X 0,Y 185.631,Z 379.543,A -85,B 0,C 180,E1 -22216.87,E2 -22216.87} C_VEL
LIN {X 0,Y 184.777,Z 381.821,A -85,B 0,C 180,E1 -22219.037,E2 -22219.037} C_VEL
LIN {X 0,Y 184.118,Z 383.673,A -85,B 0,C 180,E1 -22221.218,E2 -22221.218} C_VEL
LIN {X 0,Y 183.408,Z 385.858,A -85,B 0,C 180,E1 -22225.069,E2 -22225.069} C_VEL
LIN {X 0,Y 183.226,Z 386.656,A -85,B 0,C 180,E1 -22227.802,E2 -22227.802} C_VEL
LIN {X 0,Y 183.212,Z 386.883,A -85,B 0,C 180,E1 -22230,E2 -22230} C_VEL
LIN {X 0,Y 183.225,Z 386.689,A -85,B 0,C 180,E1 -22232.198,E2 -22232.198} C_VEL
LIN {X 0,Y 183.683,Z 385.136,A -85,B 0,C 180,E1 -22236.591,E2 -22236.591} C_VEL
LIN {X 0,Y 184.119,Z 383.779,A -85,B 0,C 180,E1 -22238.783,E2 -22238.783} C_VEL
LIN {X 0,Y 185.18,Z 380.91,A -85,B 0,C 180,E1 -22242.049,E2 -22242.049} C_VEL
LIN {X 0,Y 186.668,Z 377.019,A -85,B 0,C 180,E1 -22245.281,E2 -22245.281} C_VEL
LIN {X 0,Y 188.664,Z 371.996,A -85,B 0,C 180,E1 -22248.46,E2 -22248.46} C_VEL
LIN {X 0,Y 191.233,Z 365.666,A -85,B 0,C 180,E1 -22251.562,E2 -22251.562} C_VEL
LIN {X 0,Y 194.263,Z 357.746,A -85,B 0,C 180,E1 -22254.585,E2 -22254.585} C_VEL
LIN {X 0,Y 196.924,Z 349.797,A -85,B 0,C 180,E1 -22257.028,E2 -22257.028} C_VEL
LIN {X 0,Y 200.083,Z 339.821,A -85,B 0,C 180,E1 -22259.456,E2 -22259.456} C_VEL
LIN {X 0,Y 200.607,Z 337.553,A -85,B 0,C 180,E1 -22259.949,E2 -22259.949} C_VEL
LIN {X 0,Y 200.146,Z 328.605,A -85,B 0,C 180,E1 -22262.125,E2 -22262.125} C_VEL
LIN {X 0,Y 198.787,Z 318.063,A -85,B 0,C 180,E1 -22264.449,E2 -22264.449} C_VEL
LIN {X 0,Y 196.023,Z 306.73,A -85,B 0,C 180,E1 -22266.833,E2 -22266.833} C_VEL
LIN {X 0,Y 192.712,Z 297.368,A -85,B 0,C 180,E1 -22268.781,E2 -22268.781} C_VEL
LIN {X 0,Y 189.622,Z 290.559,A -85,B 0,C 180,E1 -22270.25,E2 -22270.25} C_VEL
LIN {X 0,Y 187.696,Z 286.917,A -85,B 0,C 180,E1 -22271.07,E2 -22271.07} C_VEL
LIN {X 0,Y 186.075,Z 283.952,A -85,B 0,C 180,E1 -22271.747,E2 -22271.747} C_VEL
LIN {X 0,Y 185.815,Z 282.833,A -85,B 0,C 180,E1 -22271.949,E2 -22271.949} C_VEL
LIN {X 0,Y 185.458,Z 280.383,A -85,B 0,C 180,E1 -22276.99,E2 -22276.99} C_VEL
LIN {X 0,Y 185.49,Z 280.381,A -85,B 0,C 180,E1 -22279.901,E2 -22279.901} C_VEL
LIN {X 0,Y 185.546,Z 280.372,A -85,B 0,C 180,E1 -22282.696,E2 -22282.696} C_VEL
LIN {X 0,Y 185.548,Z 280.371,A -85,B 0,C 180,E1 -22287.975,E2 -22287.975} C_VEL
LIN {X 0,Y 185.584,Z 280.368,A -85,B 0,C 180,E1 -22290.576,E2 -22290.576} C_VEL
LIN {X 0,Y 185.582,Z 280.366,A -85,B 0,C 180,E1 -22295.382,E2 -22295.382} C_VEL
LIN {X 0,Y 185.675,Z 280.357,A -85,B 0,C 180,E1 -22301.136,E2 -22301.136} C_VEL
LIN {X 0,Y 185.687,Z 280.355,A -85,B 0,C 180,E1 -22304.636,E2 -22304.636} C_VEL
LIN {X 0,Y 185.891,Z 280.33,A -85,B 0,C 180,E1 -22309.418,E2 -22309.418} C_VEL
LIN {X 0,Y 185.94,Z 280.322,A -85,B 0,C 180,E1 -22313.489,E2 -22313.489} C_VEL
LIN {X 0,Y 186.183,Z 280.293,A -85,B 0,C 180,E1 -22317.837,E2 -22317.837} C_VEL
LIN {X 0,Y 186.384,Z 280.267,A -85,B 0,C 180,E1 -22320,E2 -22320} C_VEL
LIN {X 0,Y 185.921,Z 280.326,A -85,B 0,C 180,E1 -22324.336,E2 -22324.336} C_VEL
LIN {X 0,Y 185.984,Z 280.319,A -85,B 0,C 180,E1 -22328.694,E2 -22328.694} C_VEL
LIN {X 0,Y 185.732,Z 280.349,A -85,B 0,C 180,E1 -22333.123,E2 -22333.123} C_VEL
LIN {X 0,Y 185.692,Z 280.353,A -85,B 0,C 180,E1 -22337.625,E2 -22337.625} C_VEL
LIN {X 0,Y 185.577,Z 280.37,A -85,B 0,C 180,E1 -22342.254,E2 -22342.254} C_VEL
LIN {X 0,Y 185.579,Z 280.368,A -85,B 0,C 180,E1 -22344.646,E2 -22344.646} C_VEL
LIN {X 0,Y 185.545,Z 280.374,A -85,B 0,C 180,E1 -22349.499,E2 -22349.499} C_VEL
LIN {X 0,Y 185.554,Z 280.553,A -85,B 0,C 180,E1 -22352.435,E2 -22352.435} C_VEL
LIN {X 0,Y 185.806,Z 281.654,A -85,B 0,C 180,E1 -22354.567,E2 -22354.567} C_VEL
LIN {X 0,Y 186.231,Z 284.709,A -85,B 0,C 180,E1 -22359.907,E2 -22359.907} C_VEL
LIN {X 0,Y 186.644,Z 287.474,A -85,B 0,C 180,E1 -22364.32,E2 -22364.32} C_VEL
LIN {X 0,Y 187.147,Z 290.332,A -85,B 0,C 180,E1 -22368.494,E2 -22368.494} C_VEL
LIN {X 0,Y 188.214,Z 293.357,A -85,B 0,C 180,E1 -22368.992,E2 -22368.992} C_VEL
LIN {X 0,Y 189.679,Z 295.918,A -85,B 0,C 180,E1 -22369.568,E2 -22369.568} C_VEL
LIN {X 0,Y 193.014,Z 303.74,A -85,B 0,C 180,E1 -22371.107,E2 -22371.107} C_VEL
LIN {X 0,Y 195.549,Z 313.353,A -85,B 0,C 180,E1 -22372.806,E2 -22372.806} C_VEL
LIN {X 0,Y 197.523,Z 324.82,A -85,B 0,C 180,E1 -22374.921,E2 -22374.921} C_VEL
LIN {X 0,Y 198.418,Z 335.876,A -85,B 0,C 180,E1 -22377.143,E2 -22377.143} C_VEL
LIN {X 0,Y 198.426,Z 345.872,A -85,B 0,C 180,E1 -22379.387,E2 -22379.387} C_VEL
LIN {X 0,Y 197.976,Z 352.642,A -85,B 0,C 180,E1 -22381.074,E2 -22381.074} C_VEL
LIN {X 0,Y 195.083,Z 361.156,A -85,B 0,C 180,E1 -22383.235,E2 -22383.235} C_VEL
LIN {X 0,Y 192.282,Z 369.015,A -85,B 0,C 180,E1 -22385.72,E2 -22385.72} C_VEL
LIN {X 0,Y 189.581,Z 376.699,A -85,B 0,C 180,E1 -22388.811,E2 -22388.811} C_VEL
LIN {X 0,Y 187.597,Z 381.965,A -85,B 0,C 180,E1 -22391.431,E2 -22391.431} C_VEL
LIN {X 0,Y 185.582,Z 387.066,A -85,B 0,C 180,E1 -22394.627,E2 -22394.627} C_VEL
LIN {X 0,Y 184.317,Z 391.036,A -85,B 0,C 180,E1 -22397.894,E2 -22397.894} C_VEL
LIN {X 0,Y 183.502,Z 393.972,A -85,B 0,C 180,E1 -22401.187,E2 -22401.187} C_VEL
LIN {X 0,Y 183.209,Z 395.37,A -85,B 0,C 180,E1 -22403.391,E2 -22403.391} C_VEL
LIN {X 0,Y 183.051,Z 396.98,A -85,B 0,C 180,E1 -22407.799,E2 -22407.799} C_VEL
LIN {X 0,Y 183.172,Z 397.196,A -85,B 0,C 180,E1 -22410,E2 -22410} C_VEL
LIN {X 0,Y 183.052,Z 396.973,A -85,B 0,C 180,E1 -22412.149,E2 -22412.149} C_VEL
LIN {X 0,Y 182.412,Z 396.592,A -85,B 0,C 180,E1 -22413.983,E2 -22413.983} C_VEL
LIN {X 0,Y 180.911,Z 395.879,A -85,B 0,C 180,E1 -22415.783,E2 -22415.783} C_VEL
LIN {X 0,Y 177.64,Z 393.582,A -85,B 0,C 180,E1 -22419.393,E2 -22419.393} C_VEL
LIN {X 0,Y 177.019,Z 392.047,A -85,B 0,C 180,E1 -22421.242,E2 -22421.242} C_VEL
LIN {X 0,Y 177.112,Z 391.468,A -85,B 0,C 180,E1 -22421.857,E2 -22421.857} C_VEL
LIN {X 0,Y 178.712,Z 386.781,A -85,B 0,C 180,E1 -22425.979,E2 -22425.979} C_VEL
LIN {X 0,Y 181.255,Z 380.654,A -85,B 0,C 180,E1 -22429.832,E2 -22429.832} C_VEL
LIN {X 0,Y 183.985,Z 373.811,A -85,B 0,C 180,E1 -22433.124,E2 -22433.124} C_VEL
LIN {X 0,Y 186.945,Z 365.662,A -85,B 0,C 180,E1 -22436.214,E2 -22436.214} C_VEL
LIN {X 0,Y 190.063,Z 357.155,A -85,B 0,C 180,E1 -22438.731,E2 -22438.731} C_VEL
LIN {X 0,Y 191.429,Z 353.241,A -85,B 0,C 180,E1 -22439.711,E2 -22439.711} C_VEL
LIN {X 0,Y 192.109,Z 342.882,A -85,B 0,C 180,E1 -22442.357,E2 -22442.357} C_VEL
LIN {X 0,Y 191.77,Z 331.411,A -85,B 0,C 180,E1 -22444.945,E2 -22444.945} C_VEL
LIN {X 0,Y 190.416,Z 320.062,A -85,B 0,C 180,E1 -22447.265,E2 -22447.265} C_VEL
LIN {X 0,Y 188.051,Z 308.646,A -85,B 0,C 180,E1 -22449.445,E2 -22449.445} C_VEL
LIN {X 0,Y 185.253,Z 301.398,A -85,B 0,C 180,E1 -22450.983,E2 -22450.983} C_VEL
LIN {X 0,Y 181.982,Z 294.617,A -85,B 0,C 180,E1 -22452.514,E2 -22452.514} C_VEL
LIN {X 0,Y 180.197,Z 291.36,A -85,B 0,C 180,E1 -22453.302,E2 -22453.302} C_VEL
LIN {X 0,Y 179.852,Z 289.976,A -85,B 0,C 180,E1 -22453.555,E2 -22453.555} C_VEL
LIN {X 0,Y 179.377,Z 287.066,A -85,B 0,C 180,E1 -22458.236,E2 -22458.236} C_VEL
LIN {X 0,Y 179.114,Z 285.047,A -85,B 0,C 180,E1 -22461.698,E2 -22461.698} C_VEL
LIN {X 0,Y 178.714,Z 282.441,A -85,B 0,C 180,E1 -22466.595,E2 -22466.595} C_VEL
LIN {X 0,Y 178.459,Z 281.261,A -85,B 0,C 180,E1 -22469.205,E2 -22469.205} C_VEL
LIN {X 0,Y 178.515,Z 281.253,A -85,B 0,C 180,E1 -22474.889,E2 -22474.889} C_VEL
LIN {X 0,Y 178.623,Z 281.236,A -85,B 0,C 180,E1 -22480.785,E2 -22480.785} C_VEL
LIN {X 0,Y 178.659,Z 281.228,A -85,B 0,C 180,E1 -22486.348,E2 -22486.348} C_VEL
LIN {X 0,Y 178.911,Z 281.199,A -85,B 0,C 180,E1 -22490.96,E2 -22490.96} C_VEL
LIN {X 0,Y 179.153,Z 281.166,A -85,B 0,C 180,E1 -22497.752,E2 -22497.752} C_VEL
LIN {X 0,Y 179.361,Z 281.143,A -85,B 0,C 180,E1 -22500,E2 -22500} C_VEL
LIN {X 0,Y 178.904,Z 281.201,A -85,B 0,C 180,E1 -22506.768,E2 -22506.768} C_VEL
LIN {X 0,Y 178.835,Z 281.209,A -85,B 0,C 180,E1 -22510.743,E2 -22510.743} C_VEL
LIN {X 0,Y 178.61,Z 281.235,A -85,B 0,C 180,E1 -22515.988,E2 -22515.988} C_VEL
LIN {X 0,Y 178.621,Z 281.235,A -85,B 0,C 180,E1 -22519.213,E2 -22519.213} C_VEL
LIN {X 0,Y 178.521,Z 281.248,A -85,B 0,C 180,E1 -22525.114,E2 -22525.114} C_VEL
LIN {X 0,Y 178.524,Z 281.247,A -85,B 0,C 180,E1 -22529.994,E2 -22529.994} C_VEL
LIN {X 0,Y 178.497,Z 281.251,A -85,B 0,C 180,E1 -22534.225,E2 -22534.225} C_VEL
LIN {X 0,Y 178.418,Z 281.258,A -85,B 0,C 180,E1 -22539.069,E2 -22539.069} C_VEL
LIN {X 0,Y 178.402,Z 281.26,A -85,B 0,C 180,E1 -22542.044,E2 -22542.044} C_VEL
LIN {X 0,Y 178.756,Z 283.334,A -85,B 0,C 180,E1 -22546.256,E2 -22546.256} C_VEL
LIN {X 0,Y 179.95,Z 286.277,A -85,B 0,C 180,E1 -22546.863,E2 -22546.863} C_VEL
LIN {X 0,Y 181.592,Z 288.724,A -85,B 0,C 180,E1 -22547.555,E2 -22547.555} C_VEL
LIN {X 0,Y 185.672,Z 296.843,A -85,B 0,C 180,E1 -22549.547,E2 -22549.547} C_VEL
LIN {X 0,Y 189.46,Z 306.815,A -85,B 0,C 180,E1 -22551.825,E2 -22551.825} C_VEL
LIN {X 0,Y 192.068,Z 317.356,A -85,B 0,C 180,E1 -22554.165,E2 -22554.165} C_VEL
LIN {X 0,Y 193.46,Z 326.341,A -85,B 0,C 180,E1 -22556.241,E2 -22556.241} C_VEL
LIN {X 0,Y 194.077,Z 336.212,A -85,B 0,C 180,E1 -22558.693,E2 -22558.693} C_VEL
LIN {X 0,Y 194.054,Z 339.433,A -85,B 0,C 180,E1 -22559.534,E2 -22559.534} C_VEL
LIN {X 0,Y 190.767,Z 349.452,A -85,B 0,C 180,E1 -22562.005,E2 -22562.005} C_VEL
LIN {X 0,Y 187.938,Z 357.539,A -85,B 0,C 180,E1 -22564.53,E2 -22564.53} C_VEL
LIN {X 0,Y 184.721,Z 365.53,A -85,B 0,C 180,E1 -22567.638,E2 -22567.638} C_VEL
LIN {X 0,Y 181.995,Z 371.94,A -85,B 0,C 180,E1 -22570.838,E2 -22570.838} C_VEL
LIN {X 0,Y 179.87,Z 377.02,A -85,B 0,C 180,E1 -22574.127,E2 -22574.127} C_VEL
LIN {X 0,Y 178.244,Z 380.963,A -85,B 0,C 180,E1 -22577.475,E2 -22577.475} C_VEL
LIN {X 0,Y 177.098,Z 383.873,A -85,B 0,C 180,E1 -22580.867,E2 -22580.867} C_VEL
LIN {X 0,Y 176.327,Z 386.161,A -85,B 0,C 180,E1 -22585.171,E2 -22585.171} C_VEL
LIN {X 0,Y 176.141,Z 386.856,A -85,B 0,C 180,E1 -22587.714,E2 -22587.714} C_VEL
LIN {X 0,Y 176.121,Z 387.082,A -85,B 0,C 180,E1 -22590,E2 -22590} C_VEL
LIN {X 0,Y 176.14,Z 386.888,A -85,B 0,C 180,E1 -22592.287,E2 -22592.287} C_VEL
LIN {X 0,Y 176.636,Z 385.335,A -85,B 0,C 180,E1 -22596.856,E2 -22596.856} C_VEL
LIN {X 0,Y 177.099,Z 383.978,A -85,B 0,C 180,E1 -22599.134,E2 -22599.134} C_VEL
LIN {X 0,Y 178.223,Z 381.11,A -85,B 0,C 180,E1 -22602.526,E2 -22602.526} C_VEL
LIN {X 0,Y 179.81,Z 377.218,A -85,B 0,C 180,E1 -22605.879,E2 -22605.879} C_VEL
LIN {X 0,Y 181.93,Z 372.195,A -85,B 0,C 180,E1 -22609.169,E2 -22609.169} C_VEL
LIN {X 0,Y 184.645,Z 365.864,A -85,B 0,C 180,E1 -22612.373,E2 -22612.373} C_VEL
LIN {X 0,Y 187.81,Z 357.944,A -85,B 0,C 180,E1 -22615.489,E2 -22615.489} C_VEL
LIN {X 0,Y 190.899,Z 349.177,A -85,B 0,C 180,E1 -22618.23,E2 -22618.23} C_VEL
LIN {X 0,Y 194.153,Z 338.967,A -85,B 0,C 180,E1 -22620.738,E2 -22620.738} C_VEL
LIN {X 0,Y 193.748,Z 329.214,A -85,B 0,C 180,E1 -22623.233,E2 -22623.233} C_VEL
LIN {X 0,Y 192.646,Z 320.051,A -85,B 0,C 180,E1 -22625.384,E2 -22625.384} C_VEL
LIN {X 0,Y 190.09,Z 308.95,A -85,B 0,C 180,E1 -22627.881,E2 -22627.881} C_VEL
LIN {X 0,Y 186.573,Z 298.841,A -85,B 0,C 180,E1 -22630.165,E2 -22630.165} C_VEL
LIN {X 0,Y 182.952,Z 291.457,A -85,B 0,C 180,E1 -22631.975,E2 -22631.975} C_VEL
LIN {X 0,Y 180.884,Z 287.539,A -85,B 0,C 180,E1 -22632.947,E2 -22632.947} C_VEL
LIN {X 0,Y 179.081,Z 284.508,A -85,B 0,C 180,E1 -22633.751,E2 -22633.751} C_VEL
LIN {X 0,Y 178.706,Z 283.105,A -85,B 0,C 180,E1 -22634.032,E2 -22634.032} C_VEL
LIN {X 0,Y 178.411,Z 281.261,A -85,B 0,C 180,E1 -22638.457,E2 -22638.457} C_VEL
LIN {X 0,Y 178.466,Z 281.256,A -85,B 0,C 180,E1 -22641.963,E2 -22641.963} C_VEL
LIN {X 0,Y 178.493,Z 281.25,A -85,B 0,C 180,E1 -22646.548,E2 -22646.548} C_VEL
LIN {X 0,Y 178.525,Z 281.246,A -85,B 0,C 180,E1 -22650.006,E2 -22650.006} C_VEL
LIN {X 0,Y 178.522,Z 281.248,A -85,B 0,C 180,E1 -22654.886,E2 -22654.886} C_VEL
LIN {X 0,Y 178.622,Z 281.234,A -85,B 0,C 180,E1 -22660.787,E2 -22660.787} C_VEL
LIN {X 0,Y 178.654,Z 281.231,A -85,B 0,C 180,E1 -22666.347,E2 -22666.347} C_VEL
LIN {X 0,Y 178.911,Z 281.198,A -85,B 0,C 180,E1 -22670.96,E2 -22670.96} C_VEL
LIN {X 0,Y 179.13,Z 281.172,A -85,B 0,C 180,E1 -22677.751,E2 -22677.751} C_VEL
LIN {X 0,Y 179.349,Z 281.144,A -85,B 0,C 180,E1 -22680,E2 -22680} C_VEL
LIN {X 0,Y 178.868,Z 281.204,A -85,B 0,C 180,E1 -22684.507,E2 -22684.507} C_VEL
LIN {X 0,Y 178.913,Z 281.199,A -85,B 0,C 180,E1 -22689.04,E2 -22689.04} C_VEL
LIN {X 0,Y 178.66,Z 281.23,A -85,B 0,C 180,E1 -22693.652,E2 -22693.652} C_VEL
LIN {X 0,Y 178.624,Z 281.233,A -85,B 0,C 180,E1 -22699.215,E2 -22699.215} C_VEL
LIN {X 0,Y 178.517,Z 281.246,A -85,B 0,C 180,E1 -22705.111,E2 -22705.111} C_VEL
LIN {X 0,Y 178.467,Z 281.317,A -85,B 0,C 180,E1 -22710.957,E2 -22710.957} C_VEL
LIN {X 0,Y 178.835,Z 282.995,A -85,B 0,C 180,E1 -22714.383,E2 -22714.383} C_VEL
LIN {X 0,Y 179.154,Z 285.44,A -85,B 0,C 180,E1 -22718.878,E2 -22718.878} C_VEL
LIN {X 0,Y 179.444,Z 287.211,A -85,B 0,C 180,E1 -22721.914,E2 -22721.914} C_VEL
LIN {X 0,Y 179.921,Z 290.215,A -85,B 0,C 180,E1 -22726.433,E2 -22726.433} C_VEL
LIN {X 0,Y 181.011,Z 293.147,A -85,B 0,C 180,E1 -22726.982,E2 -22726.982} C_VEL
LIN {X 0,Y 182.637,Z 295.736,A -85,B 0,C 180,E1 -22727.663,E2 -22727.663} C_VEL
LIN {X 0,Y 186.585,Z 304.444,A -85,B 0,C 180,E1 -22729.603,E2 -22729.603} C_VEL
LIN {X 0,Y 188.703,Z 311.072,A -85,B 0,C 180,E1 -22730.943,E2 -22730.943} C_VEL
LIN {X 0,Y 190.768,Z 321.957,A -85,B 0,C 180,E1 -22733.042,E2 -22733.042} C_VEL
LIN {X 0,Y 191.897,Z 332.675,A -85,B 0,C 180,E1 -22735.255,E2 -22735.255} C_VEL
LIN {X 0,Y 192.131,Z 343.085,A -85,B 0,C 180,E1 -22737.62,E2 -22737.62} C_VEL
LIN {X 0,Y 191.566,Z 352.438,A -85,B 0,C 180,E1 -22740.009,E2 -22740.009} C_VEL
LIN {X 0,Y 190.088,Z 357.379,A -85,B 0,C 180,E1 -22741.272,E2 -22741.272} C_VEL
LIN {X 0,Y 186.931,Z 365.838,A -85,B 0,C 180,E1 -22743.783,E2 -22743.783} C_VEL
LIN {X 0,Y 184.325,Z 372.948,A -85,B 0,C 180,E1 -22746.437,E2 -22746.437} C_VEL
LIN {X 0,Y 181.618,Z 379.757,A -85,B 0,C 180,E1 -22749.618,E2 -22749.618} C_VEL
LIN {X 0,Y 179.372,Z 385.278,A -85,B 0,C 180,E1 -22752.911,E2 -22752.911} C_VEL
LIN {X 0,Y 177.767,Z 389.613,A -85,B 0,C 180,E1 -22756.278,E2 -22756.278} C_VEL
LIN {X 0,Y 176.995,Z 391.911,A -85,B 0,C 180,E1 -22758.548,E2 -22758.548} C_VEL
LIN {X 0,Y 176.462,Z 393.772,A -85,B 0,C 180,E1 -22760.833,E2 -22760.833} C_VEL
LIN {X 0,Y 176.137,Z 395.17,A -85,B 0,C 180,E1 -22763.125,E2 -22763.125} C_VEL
LIN {X 0,Y 175.969,Z 396.781,A -85,B 0,C 180,E1 -22767.711,E2 -22767.711} C_VEL
LIN {X 0,Y 176.079,Z 396.996,A -85,B 0,C 180,E1 -22770,E2 -22770} C_VEL
LIN {X 0,Y 175.947,Z 396.608,A -85,B 0,C 180,E1 -22773.037,E2 -22773.037} C_VEL
LIN {X 0,Y 176.115,Z 395.14,A -85,B 0,C 180,E1 -22776.876,E2 -22776.876} C_VEL
LIN {X 0,Y 176.457,Z 393.729,A -85,B 0,C 180,E1 -22779.167,E2 -22779.167} C_VEL
LIN {X 0,Y 177.112,Z 391.468,A -85,B 0,C 180,E1 -22781.857,E2 -22781.857} C_VEL
LIN {X 0,Y 177.068,Z 389.646,A -85,B 0,C 180,E1 -22783.676,E2 -22783.676} C_VEL
LIN {X 0,Y 175.532,Z 386.202,A -85,B 0,C 180,E1 -22786.661,E2 -22786.661} C_VEL
LIN {X 0,Y 174.409,Z 382.122,A -85,B 0,C 180,E1 -22789.601,E2 -22789.601} C_VEL
LIN {X 0,Y 175,Z 379.267,A -85,B 0,C 180,E1 -22791.29,E2 -22791.29} C_VEL
LIN {X 0,Y 177.775,Z 372.788,A -85,B 0,C 180,E1 -22794.392,E2 -22794.392} C_VEL
LIN {X 0,Y 180.571,Z 365.459,A -85,B 0,C 180,E1 -22797.214,E2 -22797.214} C_VEL
LIN {X 0,Y 183.861,Z 356.952,A -85,B 0,C 180,E1 -22799.796,E2 -22799.796} C_VEL
LIN {X 0,Y 185,Z 353.029,A -85,B 0,C 180,E1 -22800.854,E2 -22800.854} C_VEL
LIN {X 0,Y 185.711,Z 343.877,A -85,B 0,C 180,E1 -22803.312,E2 -22803.312} C_VEL
LIN {X 0,Y 185.544,Z 332.597,A -85,B 0,C 180,E1 -22806.004,E2 -22806.004} C_VEL
LIN {X 0,Y 184.4,Z 321.736,A -85,B 0,C 180,E1 -22808.371,E2 -22808.371} C_VEL
LIN {X 0,Y 182.335,Z 311.157,A -85,B 0,C 180,E1 -22810.56,E2 -22810.56} C_VEL
LIN {X 0,Y 179.089,Z 302.932,A -85,B 0,C 180,E1 -22812.521,E2 -22812.521} C_VEL
LIN {X 0,Y 177.043,Z 298.781,A -85,B 0,C 180,E1 -22813.576,E2 -22813.576} C_VEL
LIN {X 0,Y 174.902,Z 294.526,A -85,B 0,C 180,E1 -22814.66,E2 -22814.66} C_VEL
LIN {X 0,Y 173.041,Z 291.339,A -85,B 0,C 180,E1 -22815.553,E2 -22815.553} C_VEL
LIN {X 0,Y 172.585,Z 289.713,A -85,B 0,C 180,E1 -22815.906,E2 -22815.906} C_VEL
LIN {X 0,Y 172.179,Z 286.852,A -85,B 0,C 180,E1 -22820.854,E2 -22820.854} C_VEL
LIN {X 0,Y 171.898,Z 284.623,A -85,B 0,C 180,E1 -22825.083,E2 -22825.083} C_VEL
LIN {X 0,Y 171.408,Z 282.14,A -85,B 0,C 180,E1 -22830.527,E2 -22830.527} C_VEL
LIN {X 0,Y 171.442,Z 282.133,A -85,B 0,C 180,E1 -22835.799,E2 -22835.799} C_VEL
LIN {X 0,Y 171.579,Z 282.113,A -85,B 0,C 180,E1 -22840.872,E2 -22840.872} C_VEL
LIN {X 0,Y 171.577,Z 282.112,A -85,B 0,C 180,E1 -22845.773,E2 -22845.773} C_VEL
LIN {X 0,Y 171.848,Z 282.079,A -85,B 0,C 180,E1 -22850.585,E2 -22850.585} C_VEL
LIN {X 0,Y 171.815,Z 282.081,A -85,B 0,C 180,E1 -22855.308,E2 -22855.308} C_VEL
LIN {X 0,Y 172.324,Z 282.02,A -85,B 0,C 180,E1 -22860,E2 -22860} C_VEL
LIN {X 0,Y 171.866,Z 282.077,A -85,B 0,C 180,E1 -22867.047,E2 -22867.047} C_VEL
LIN {X 0,Y 171.769,Z 282.088,A -85,B 0,C 180,E1 -22870.896,E2 -22870.896} C_VEL
LIN {X 0,Y 171.546,Z 282.117,A -85,B 0,C 180,E1 -22876.666,E2 -22876.666} C_VEL
LIN {X 0,Y 171.54,Z 282.117,A -85,B 0,C 180,E1 -22879.557,E2 -22879.557} C_VEL
LIN {X 0,Y 171.46,Z 282.128,A -85,B 0,C 180,E1 -22885.61,E2 -22885.61} C_VEL
LIN {X 0,Y 171.443,Z 282.13,A -85,B 0,C 180,E1 -22890.587,E2 -22890.587} C_VEL
LIN {X 0,Y 171.408,Z 282.134,A -85,B 0,C 180,E1 -22895.032,E2 -22895.032} C_VEL
LIN {X 0,Y 171.38,Z 282.136,A -85,B 0,C 180,E1 -22898.817,E2 -22898.817} C_VEL
LIN {X 0,Y 171.344,Z 282.174,A -85,B 0,C 180,E1 -22901.016,E2 -22901.016} C_VEL
LIN {X 0,Y 171.546,Z 283.506,A -85,B 0,C 180,E1 -22903.894,E2 -22903.894} C_VEL
LIN {X 0,Y 172.712,Z 286.353,A -85,B 0,C 180,E1 -22904.548,E2 -22904.548} C_VEL
LIN {X 0,Y 174.641,Z 289.138,A -85,B 0,C 180,E1 -22905.444,E2 -22905.444} C_VEL
LIN {X 0,Y 179.205,Z 297.866,A -85,B 0,C 180,E1 -22907.856,E2 -22907.856} C_VEL
LIN {X 0,Y 182.541,Z 306.012,A -85,B 0,C 180,E1 -22909.925,E2 -22909.925} C_VEL
LIN {X 0,Y 184.996,Z 314.576,A -85,B 0,C 180,E1 -22911.996,E2 -22911.996} C_VEL
LIN {X 0,Y 186.866,Z 324.594,A -85,B 0,C 180,E1 -22914.439,E2 -22914.439} C_VEL
LIN {X 0,Y 187.62,Z 334.33,A -85,B 0,C 180,E1 -22916.925,E2 -22916.925} C_VEL
LIN {X 0,Y 187.622,Z 340.707,A -85,B 0,C 180,E1 -22918.686,E2 -22918.686} C_VEL
LIN {X 0,Y 183.99,Z 351.102,A -85,B 0,C 180,E1 -22921.387,E2 -22921.387} C_VEL
LIN {X 0,Y 180.996,Z 359.22,A -85,B 0,C 180,E1 -22924.098,E2 -22924.098} C_VEL
LIN {X 0,Y 177.665,Z 366.898,A -85,B 0,C 180,E1 -22927.314,E2 -22927.314} C_VEL
LIN {X 0,Y 174.485,Z 373.948,A -85,B 0,C 180,E1 -22931.202,E2 -22931.202} C_VEL
LIN {X 0,Y 172.381,Z 378.638,A -85,B 0,C 180,E1 -22934.633,E2 -22934.633} C_VEL
LIN {X 0,Y 170.869,Z 382.222,A -85,B 0,C 180,E1 -22938.132,E2 -22938.132} C_VEL
LIN {X 0,Y 170.103,Z 384.073,A -85,B 0,C 180,E1 -22940.488,E2 -22940.488} C_VEL
LIN {X 0,Y 169.585,Z 385.462,A -85,B 0,C 180,E1 -22942.858,E2 -22942.858} C_VEL
LIN {X 0,Y 169.056,Z 387.056,A -85,B 0,C 180,E1 -22947.618,E2 -22947.618} C_VEL
LIN {X 0,Y 169.032,Z 387.282,A -85,B 0,C 180,E1 -22950,E2 -22950} C_VEL
LIN {X 0,Y 169.194,Z 386.591,A -85,B 0,C 180,E1 -22954.497,E2 -22954.497} C_VEL
LIN {X 0,Y 169.585,Z 385.534,A -85,B 0,C 180,E1 -22957.142,E2 -22957.142} C_VEL
LIN {X 0,Y 170.103,Z 384.177,A -85,B 0,C 180,E1 -22959.513,E2 -22959.513} C_VEL
LIN {X 0,Y 171.294,Z 381.309,A -85,B 0,C 180,E1 -22963.042,E2 -22963.042} C_VEL
LIN {X 0,Y 172.982,Z 377.417,A -85,B 0,C 180,E1 -22966.523,E2 -22966.523} C_VEL
LIN {X 0,Y 175.235,Z 372.394,A -85,B 0,C 180,E1 -22969.932,E2 -22969.932} C_VEL
LIN {X 0,Y 178.096,Z 366.062,A -85,B 0,C 180,E1 -22973.243,E2 -22973.243} C_VEL
LIN {X 0,Y 181.41,Z 358.141,A -85,B 0,C 180,E1 -22976.457,E2 -22976.457} C_VEL
LIN {X 0,Y 184.441,Z 349.988,A -85,B 0,C 180,E1 -22979.096,E2 -22979.096} C_VEL
LIN {X 0,Y 187.475,Z 341.28,A -85,B 0,C 180,E1 -22981.342,E2 -22981.342} C_VEL
LIN {X 0,Y 187.736,Z 336.324,A -85,B 0,C 180,E1 -22982.691,E2 -22982.691} C_VEL
LIN {X 0,Y 187.087,Z 325.952,A -85,B 0,C 180,E1 -22985.391,E2 -22985.391} C_VEL
LIN {X 0,Y 185.248,Z 315.599,A -85,B 0,C 180,E1 -22987.943,E2 -22987.943} C_VEL
LIN {X 0,Y 182.709,Z 306.513,A -85,B 0,C 180,E1 -22990.137,E2 -22990.137} C_VEL
LIN {X 0,Y 179.307,Z 298.065,A -85,B 0,C 180,E1 -22992.284,E2 -22992.284} C_VEL
LIN {X 0,Y 176.24,Z 292.142,A -85,B 0,C 180,E1 -22993.922,E2 -22993.922} C_VEL
LIN {X 0,Y 173.964,Z 288.032,A -85,B 0,C 180,E1 -22995.084,E2 -22995.084} C_VEL
LIN {X 0,Y 172.03,Z 285.106,A -85,B 0,C 180,E1 -22996.012,E2 -22996.012} C_VEL
LIN {X 0,Y 171.511,Z 283.364,A -85,B 0,C 180,E1 -22996.406,E2 -22996.406} C_VEL
LIN {X 0,Y 171.377,Z 282.265,A -85,B 0,C 180,E1 -22998.993,E2 -22998.993} C_VEL
LIN {X 0,Y 171.415,Z 282.134,A -85,B 0,C 180,E1 -23002.048,E2 -23002.048} C_VEL
LIN {X 0,Y 171.413,Z 282.133,A -85,B 0,C 180,E1 -23005.086,E2 -23005.086} C_VEL
LIN {X 0,Y 171.452,Z 282.129,A -85,B 0,C 180,E1 -23010.535,E2 -23010.535} C_VEL
LIN {X 0,Y 171.446,Z 282.123,A -85,B 0,C 180,E1 -23015.8,E2 -23015.8} C_VEL
LIN {X 0,Y 171.578,Z 282.112,A -85,B 0,C 180,E1 -23020.871,E2 -23020.871} C_VEL
LIN {X 0,Y 171.571,Z 282.113,A -85,B 0,C 180,E1 -23025.772,E2 -23025.772} C_VEL
LIN {X 0,Y 171.848,Z 282.077,A -85,B 0,C 180,E1 -23030.585,E2 -23030.585} C_VEL
LIN {X 0,Y 171.794,Z 282.086,A -85,B 0,C 180,E1 -23035.307,E2 -23035.307} C_VEL
LIN {X 0,Y 172.314,Z 282.02,A -85,B 0,C 180,E1 -23040,E2 -23040} C_VEL
LIN {X 0,Y 171.816,Z 282.082,A -85,B 0,C 180,E1 -23044.692,E2 -23044.692} C_VEL
LIN {X 0,Y 171.849,Z 282.078,A -85,B 0,C 180,E1 -23049.415,E2 -23049.415} C_VEL
LIN {X 0,Y 171.578,Z 282.113,A -85,B 0,C 180,E1 -23054.227,E2 -23054.227} C_VEL
LIN {X 0,Y 171.543,Z 282.115,A -85,B 0,C 180,E1 -23059.559,E2 -23059.559} C_VEL
LIN {X 0,Y 171.444,Z 282.124,A -85,B 0,C 180,E1 -23065.597,E2 -23065.597} C_VEL
LIN {X 0,Y 171.414,Z 282.15,A -85,B 0,C 180,E1 -23069.472,E2 -23069.472} C_VEL
LIN {X 0,Y 171.658,Z 283.356,A -85,B 0,C 180,E1 -23072.157,E2 -23072.157} C_VEL
LIN {X 0,Y 171.905,Z 284.809,A -85,B 0,C 180,E1 -23075.148,E2 -23075.148} C_VEL
LIN {X 0,Y 172.307,Z 287.815,A -85,B 0,C 180,E1 -23080.738,E2 -23080.738} C_VEL
LIN {X 0,Y 172.641,Z 289.833,A -85,B 0,C 180,E1 -23084.08,E2 -23084.08} C_VEL
LIN {X 0,Y 173.787,Z 292.908,A -85,B 0,C 180,E1 -23084.72,E2 -23084.72} C_VEL
LIN {X 0,Y 175.598,Z 295.695,A -85,B 0,C 180,E1 -23085.552,E2 -23085.552} C_VEL
LIN {X 0,Y 177.707,Z 299.737,A -85,B 0,C 180,E1 -23086.618,E2 -23086.618} C_VEL
LIN {X 0,Y 181.001,Z 307.303,A -85,B 0,C 180,E1 -23088.453,E2 -23088.453} C_VEL
LIN {X 0,Y 182.903,Z 313.116,A -85,B 0,C 180,E1 -23089.764,E2 -23089.764} C_VEL
LIN {X 0,Y 184.849,Z 324.395,A -85,B 0,C 180,E1 -23092.114,E2 -23092.114} C_VEL
LIN {X 0,Y 185.735,Z 335.388,A -85,B 0,C 180,E1 -23094.563,E2 -23094.563} C_VEL
LIN {X 0,Y 185.713,Z 345.197,A -85,B 0,C 180,E1 -23096.965,E2 -23096.965} C_VEL
LIN {X 0,Y 185.075,Z 353.275,A -85,B 0,C 180,E1 -23099.159,E2 -23099.159} C_VEL
LIN {X 0,Y 183.194,Z 358.975,A -85,B 0,C 180,E1 -23100.716,E2 -23100.716} C_VEL
LIN {X 0,Y 179.946,Z 367.13,A -85,B 0,C 180,E1 -23103.311,E2 -23103.311} C_VEL
LIN {X 0,Y 177.577,Z 373.31,A -85,B 0,C 180,E1 -23105.766,E2 -23105.766} C_VEL
LIN {X 0,Y 174.548,Z 380.572,A -85,B 0,C 180,E1 -23109.371,E2 -23109.371} C_VEL
LIN {X 0,Y 171.874,Z 386.667,A -85,B 0,C 180,E1 -23113.367,E2 -23113.367} C_VEL
LIN {X 0,Y 170.401,Z 390.637,A -85,B 0,C 180,E1 -23116.889,E2 -23116.889} C_VEL
LIN {X 0,Y 169.42,Z 393.572,A -85,B 0,C 180,E1 -23120.448,E2 -23120.448} C_VEL
LIN {X 0,Y 169.072,Z 394.97,A -85,B 0,C 180,E1 -23122.836,E2 -23122.836} C_VEL
LIN {X 0,Y 168.86,Z 396.581,A -85,B 0,C 180,E1 -23127.614,E2 -23127.614} C_VEL
LIN {X 0,Y 168.988,Z 396.796,A -85,B 0,C 180,E1 -23130,E2 -23130} C_VEL
LIN {X 0,Y 168.857,Z 396.507,A -85,B 0,C 180,E1 -23132.679,E2 -23132.679} C_VEL
LIN {X 0,Y 169.04,Z 394.939,A -85,B 0,C 180,E1 -23137.165,E2 -23137.165} C_VEL
LIN {X 0,Y 169.416,Z 393.528,A -85,B 0,C 180,E1 -23139.551,E2 -23139.551} C_VEL
LIN {X 0,Y 170.401,Z 390.573,A -85,B 0,C 180,E1 -23143.111,E2 -23143.111} C_VEL
LIN {X 0,Y 171.872,Z 386.579,A -85,B 0,C 180,E1 -23146.633,E2 -23146.633} C_VEL
LIN {X 0,Y 174.537,Z 380.451,A -85,B 0,C 180,E1 -23150.63,E2 -23150.63} C_VEL
LIN {X 0,Y 175,Z 379.267,A -85,B 0,C 180,E1 -23151.29,E2 -23151.29} C_VEL
LIN {X 0,Y 175.69,Z 376.222,A -85,B 0,C 180,E1 -23152.929,E2 -23152.929} C_VEL
LIN {X 0,Y 175.234,Z 370.892,A -85,B 0,C 180,E1 -23155.66,E2 -23155.66} C_VEL
LIN {X 0,Y 175.004,Z 365.014,A -85,B 0,C 180,E1 -23158.269,E2 -23158.269} C_VEL
LIN {X 0,Y 176.008,Z 361.044,A -85,B 0,C 180,E1 -23159.667,E2 -23159.667} C_VEL
LIN {X 0,Y 178.346,Z 354.792,A -85,B 0,C 180,E1 -23161.476,E2 -23161.476} C_VEL
LIN {X 0,Y 179.368,Z 344.804,A -85,B 0,C 180,E1 -23164.329,E2 -23164.329} C_VEL
LIN {X 0,Y 179.36,Z 333.825,A -85,B 0,C 180,E1 -23167.132,E2 -23167.132} C_VEL
LIN {X 0,Y 178.418,Z 323.021,A -85,B 0,C 180,E1 -23169.633,E2 -23169.633} C_VEL
LIN {X 0,Y 176.986,Z 314.862,A -85,B 0,C 180,E1 -23171.452,E2 -23171.452} C_VEL
LIN {X 0,Y 174.079,Z 307.005,A -85,B 0,C 180,E1 -23173.494,E2 -23173.494} C_VEL
LIN {X 0,Y 171.962,Z 302.507,A -85,B 0,C 180,E1 -23174.756,E2 -23174.756} C_VEL
LIN {X 0,Y 170.374,Z 299.207,A -85,B 0,C 180,E1 -23175.67,E2 -23175.67} C_VEL
LIN {X 0,Y 168.402,Z 295.225,A -85,B 0,C 180,E1 -23176.796,E2 -23176.796} C_VEL
LIN {X 0,Y 165.989,Z 291.568,A -85,B 0,C 180,E1 -23178.04,E2 -23178.04} C_VEL
LIN {X 0,Y 165.362,Z 289.437,A -85,B 0,C 180,E1 -23178.525,E2 -23178.525} C_VEL
LIN {X 0,Y 164.978,Z 286.54,A -85,B 0,C 180,E1 -23184.037,E2 -23184.037} C_VEL
LIN {X 0,Y 164.568,Z 284.174,A -85,B 0,C 180,E1 -23189.172,E2 -23189.172} C_VEL
LIN {X 0,Y 164.309,Z 283.034,A -85,B 0,C 180,E1 -23191.933,E2 -23191.933} C_VEL
LIN {X 0,Y 164.394,Z 283.011,A -85,B 0,C 180,E1 -23194.69,E2 -23194.69} C_VEL
LIN {X 0,Y 164.485,Z 282.996,A -85,B 0,C 180,E1 -23200.052,E2 -23200.052} C_VEL
LIN {X 0,Y 164.525,Z 282.991,A -85,B 0,C 180,E1 -23205.149,E2 -23205.149} C_VEL
LIN {X 0,Y 164.768,Z 282.961,A -85,B 0,C 180,E1 -23210.176,E2 -23210.176} C_VEL
LIN {X 0,Y 164.831,Z 282.951,A -85,B 0,C 180,E1 -23212.651,E2 -23212.651} C_VEL
LIN {X 0,Y 165.048,Z 282.924,A -85,B 0,C 180,E1 -23217.56,E2 -23217.56} C_VEL
LIN {X 0,Y 165.287,Z 282.896,A -85,B 0,C 180,E1 -23220,E2 -23220} C_VEL
LIN {X 0,Y 164.827,Z 282.953,A -85,B 0,C 180,E1 -23227.349,E2 -23227.349} C_VEL
LIN {X 0,Y 164.703,Z 282.967,A -85,B 0,C 180,E1 -23231.061,E2 -23231.061} C_VEL
LIN {X 0,Y 164.477,Z 282.996,A -85,B 0,C 180,E1 -23237.404,E2 -23237.404} C_VEL
LIN {X 0,Y 164.473,Z 282.998,A -85,B 0,C 180,E1 -23239.989,E2 -23239.989} C_VEL
LIN {X 0,Y 164.387,Z 283.008,A -85,B 0,C 180,E1 -23246.129,E2 -23246.129} C_VEL
LIN {X 0,Y 164.377,Z 283.008,A -85,B 0,C 180,E1 -23251.229,E2 -23251.229} C_VEL
LIN {X 0,Y 164.314,Z 283.018,A -85,B 0,C 180,E1 -23256.785,E2 -23256.785} C_VEL
LIN {X 0,Y 164.317,Z 283.156,A -85,B 0,C 180,E1 -23259.909,E2 -23259.909} C_VEL
LIN {X 0,Y 164.408,Z 283.649,A -85,B 0,C 180,E1 -23261.192,E2 -23261.192} C_VEL
LIN {X 0,Y 165.665,Z 286.799,A -85,B 0,C 180,E1 -23262.028,E2 -23262.028} C_VEL
LIN {X 0,Y 167.677,Z 289.53,A -85,B 0,C 180,E1 -23263.06,E2 -23263.06} C_VEL
LIN {X 0,Y 169.687,Z 293.054,A -85,B 0,C 180,E1 -23264.199,E2 -23264.199} C_VEL
LIN {X 0,Y 173.88,Z 301.226,A -85,B 0,C 180,E1 -23266.681,E2 -23266.681} C_VEL
LIN {X 0,Y 177.059,Z 309.396,A -85,B 0,C 180,E1 -23268.953,E2 -23268.953} C_VEL
LIN {X 0,Y 179.098,Z 316.806,A -85,B 0,C 180,E1 -23270.896,E2 -23270.896} C_VEL
LIN {X 0,Y 180.839,Z 327.314,A -85,B 0,C 180,E1 -23273.654,E2 -23273.654} C_VEL
LIN {X 0,Y 181.326,Z 336.531,A -85,B 0,C 180,E1 -23276.176,E2 -23276.176} C_VEL
LIN {X 0,Y 181.237,Z 341.975,A -85,B 0,C 180,E1 -23277.778,E2 -23277.778} C_VEL
LIN {X 0,Y 177.548,Z 351.925,A -85,B 0,C 180,E1 -23280.474,E2 -23280.474} C_VEL
LIN {X 0,Y 173.969,Z 360.807,A -85,B 0,C 180,E1 -23283.617,E2 -23283.617} C_VEL
LIN {X 0,Y 170.599,Z 368.211,A -85,B 0,C 180,E1 -23286.961,E2 -23286.961} C_VEL
LIN {X 0,Y 167.76,Z 374.15,A -85,B 0,C 180,E1 -23290.419,E2 -23290.419} C_VEL
LIN {X 0,Y 165.541,Z 378.839,A -85,B 0,C 180,E1 -23293.981,E2 -23293.981} C_VEL
LIN {X 0,Y 163.918,Z 382.423,A -85,B 0,C 180,E1 -23297.621,E2 -23297.621} C_VEL
LIN {X 0,Y 163.092,Z 384.274,A -85,B 0,C 180,E1 -23300.075,E2 -23300.075} C_VEL
LIN {X 0,Y 162.548,Z 385.662,A -85,B 0,C 180,E1 -23302.547,E2 -23302.547} C_VEL
LIN {X 0,Y 161.975,Z 387.256,A -85,B 0,C 180,E1 -23307.513,E2 -23307.513} C_VEL
LIN {X 0,Y 161.945,Z 387.481,A -85,B 0,C 180,E1 -23310,E2 -23310} C_VEL
LIN {X 0,Y 162.067,Z 386.964,A -85,B 0,C 180,E1 -23314.137,E2 -23314.137} C_VEL
LIN {X 0,Y 162.548,Z 385.734,A -85,B 0,C 180,E1 -23317.453,E2 -23317.453} C_VEL
LIN {X 0,Y 163.092,Z 384.377,A -85,B 0,C 180,E1 -23319.926,E2 -23319.926} C_VEL
LIN {X 0,Y 164.391,Z 381.507,A -85,B 0,C 180,E1 -23323.6,E2 -23323.6} C_VEL
LIN {X 0,Y 166.186,Z 377.616,A -85,B 0,C 180,E1 -23327.22,E2 -23327.22} C_VEL
LIN {X 0,Y 168.578,Z 372.592,A -85,B 0,C 180,E1 -23330.755,E2 -23330.755} C_VEL
LIN {X 0,Y 171.595,Z 366.26,A -85,B 0,C 180,E1 -23334.178,E2 -23334.178} C_VEL
LIN {X 0,Y 175.076,Z 358.339,A -85,B 0,C 180,E1 -23337.493,E2 -23337.493} C_VEL
LIN {X 0,Y 178.933,Z 348.489,A -85,B 0,C 180,E1 -23340.704,E2 -23340.704} C_VEL
LIN {X 0,Y 181.338,Z 341.48,A -85,B 0,C 180,E1 -23342.531,E2 -23342.531} C_VEL
LIN {X 0,Y 181.273,Z 332.673,A -85,B 0,C 180,E1 -23345.068,E2 -23345.068} C_VEL
LIN {X 0,Y 180.553,Z 324.899,A -85,B 0,C 180,E1 -23347.171,E2 -23347.171} C_VEL
LIN {X 0,Y 178.601,Z 314.689,A -85,B 0,C 180,E1 -23349.839,E2 -23349.839} C_VEL
LIN {X 0,Y 175.739,Z 305.563,A -85,B 0,C 180,E1 -23352.284,E2 -23352.284} C_VEL
LIN {X 0,Y 171.893,Z 297.167,A -85,B 0,C 180,E1 -23354.733,E2 -23354.733} C_VEL
LIN {X 0,Y 169.543,Z 292.881,A -85,B 0,C 180,E1 -23356.086,E2 -23356.086} C_VEL
LIN {X 0,Y 167.604,Z 289.37,A -85,B 0,C 180,E1 -23357.201,E2 -23357.201} C_VEL
LIN {X 0,Y 165,Z 285.568,A -85,B 0,C 180,E1 -23358.583,E2 -23358.583} C_VEL
LIN {X 0,Y 164.429,Z 283.66,A -85,B 0,C 180,E1 -23359.018,E2 -23359.018} C_VEL
LIN {X 0,Y 164.329,Z 283.156,A -85,B 0,C 180,E1 -23360.338,E2 -23360.338} C_VEL
LIN {X 0,Y 164.346,Z 283.014,A -85,B 0,C 180,E1 -23364.342,E2 -23364.342} C_VEL
LIN {X 0,Y 164.393,Z 283.003,A -85,B 0,C 180,E1 -23369.135,E2 -23369.135} C_VEL
LIN {X 0,Y 164.409,Z 283.006,A -85,B 0,C 180,E1 -23374.693,E2 -23374.693} C_VEL
LIN {X 0,Y 164.486,Z 282.994,A -85,B 0,C 180,E1 -23380.052,E2 -23380.052} C_VEL
LIN {X 0,Y 164.501,Z 282.993,A -85,B 0,C 180,E1 -23385.147,E2 -23385.147} C_VEL
LIN {X 0,Y 164.769,Z 282.96,A -85,B 0,C 180,E1 -23390.176,E2 -23390.176} C_VEL
LIN {X 0,Y 164.827,Z 282.954,A -85,B 0,C 180,E1 -23392.651,E2 -23392.651} C_VEL
LIN {X 0,Y 165.278,Z 282.897,A -85,B 0,C 180,E1 -23400,E2 -23400} C_VEL
LIN {X 0,Y 164.765,Z 282.96,A -85,B 0,C 180,E1 -23404.894,E2 -23404.894} C_VEL
LIN {X 0,Y 164.832,Z 282.951,A -85,B 0,C 180,E1 -23407.349,E2 -23407.349} C_VEL
LIN {X 0,Y 164.705,Z 282.969,A -85,B 0,C 180,E1 -23411.061,E2 -23411.061} C_VEL
LIN {X 0,Y 164.485,Z 282.994,A -85,B 0,C 180,E1 -23417.403,E2 -23417.403} C_VEL
LIN {X 0,Y 164.475,Z 282.997,A -85,B 0,C 180,E1 -23419.989,E2 -23419.989} C_VEL
LIN {X 0,Y 164.371,Z 283.005,A -85,B 0,C 180,E1 -23426.116,E2 -23426.116} C_VEL
LIN {X 0,Y 164.335,Z 283.094,A -85,B 0,C 180,E1 -23428.062,E2 -23428.062} C_VEL
LIN {X 0,Y 164.635,Z 284.478,A -85,B 0,C 180,E1 -23431.375,E2 -23431.375} C_VEL
LIN {X 0,Y 165.012,Z 286.925,A -85,B 0,C 180,E1 -23436.603,E2 -23436.603} C_VEL
LIN {X 0,Y 165.367,Z 289.448,A -85,B 0,C 180,E1 -23441.379,E2 -23441.379} C_VEL
LIN {X 0,Y 166.469,Z 292.5,A -85,B 0,C 180,E1 -23442.103,E2 -23442.103} C_VEL
LIN {X 0,Y 168.561,Z 295.595,A -85,B 0,C 180,E1 -23443.172,E2 -23443.172} C_VEL
LIN {X 0,Y 170.605,Z 299.495,A -85,B 0,C 180,E1 -23444.323,E2 -23444.323} C_VEL
LIN {X 0,Y 174.957,Z 308.858,A -85,B 0,C 180,E1 -23446.93,E2 -23446.93} C_VEL
LIN {X 0,Y 177.403,Z 316.455,A -85,B 0,C 180,E1 -23448.825,E2 -23448.825} C_VEL
LIN {X 0,Y 178.998,Z 327.748,A -85,B 0,C 180,E1 -23451.363,E2 -23451.363} C_VEL
